// TwinCAT 3 PLC project Samples
// Title: BA2_Templates
// Company: Beckhoff Automation GmbH
// Author: Beckhoff Automation GmbH
// ProjectVersion: 2.2.0.0
// Description: Library that covers all technical building automation services in a built-in skeleton. It contains function blocks for conventional HVAC and room automation.
// ProgramVersion: 3.1.4026.20
// libraries:
//   Tc2_MDP, * (Beckhoff Automation GmbH)
//   Tc2_SerialCom, * (Beckhoff Automation GmbH)
//   Tc2_Standard, * (Beckhoff Automation GmbH)
//   Tc2_SUPS, * (Beckhoff Automation GmbH)
//   Tc2_System, * (Beckhoff Automation GmbH)
//   Tc2_Utilities, * (Beckhoff Automation GmbH)
//   Tc3_BA2, * (Beckhoff Automation GmbH)
//   Tc3_BA2_Common, * (Beckhoff Automation GmbH)
//   Tc3_BACnetRev14, * (Beckhoff Automation GmbH)
//   Tc3_DALI, * (Beckhoff Automation GmbH)
//   Tc3_Module, * (Beckhoff Automation GmbH)
//   Tc3_XBA, * (Beckhoff Automation GmbH)
// project tree:
//   / FastTask.TcTTO, PlcTask.TcTTO (not stored)
//   POUs/ DALICommunication.TcPOU, MAIN.TcPOU
//   Templates/DUTs/Enumerations/Building/ E_BA_BuildingMode.TcDUT (not stored)
//   Templates/DUTs/Enumerations/Plant/AC/ E_BA_AC_OpMod01.TcDUT (not stored), E_BA_AC_OpMod02.TcDUT, E_BA_AC_PlantStep01.TcDUT (not stored), E_BA_AC_SelSpErc.TcDUT, E_BA_AC_SeqNumber_H.TcDUT (not stored), E_BA_AC_SeqNumber_T.TcDUT (not stored)
//   Templates/DUTs/Enumerations/Process/ E_BA_Process.TcDUT (not stored)
//   Templates/DUTs/Enumerations/System/ E_BA_UPSType.TcDUT (not stored)
//   Templates/DUTs/Enumerations/Universal/ E_BA_3Point.TcDUT (not stored), E_BA_3PointA.TcDUT, E_BA_3Step.TcDUT, E_BA_3StepA.TcDUT, E_BA_Conversion_kFactor.TcDUT (not stored), E_BA_EnergyLvl.TcDUT (not stored), E_BA_EnergyLvlA.TcDUT, E_BA_EnergyLvlEx.TcDUT, E_BA_EnergyLvlExA.TcDUT, E_BA_OnOff.TcDUT, E_BA_OnOffA.TcDUT (not stored)
//   Templates/DUTs/Types/Actuator/ ST_BA_LightActuatorFeedback.TcDUT (not stored), ST_BA_SunblindActuatorFeedback.TcDUT (not stored)
//   Templates/DUTs/Types/Building/ ST_BA_BuildingAlarms.TcDUT (not stored), ST_BA_BuildingLighting.TcDUT, ST_BA_BuildingSunblind.TcDUT (not stored)
//   Templates/DUTs/Types/Facade/ ST_BA_Facade.TcDUT (not stored)
//   Templates/DUTs/Types/General/ ST_BA_GeneralSettings.TcDUT (not stored), ST_BA_GlobalAlarmsEvents.TcDUT
//   Templates/DUTs/Types/WeatherStation/ ST_BA_WeatherStation.TcDUT (not stored), ST_BA_WSC11Data.TcDUT, ST_BA_WSC11Status.TcDUT (not stored)
//   Templates/GVLs/ BA2_Param.TcGVL, LblComp.TcGVL, Priority.TcGVL (not stored), SysTime.TcGVL
//   Templates/GVLs/EventClassesID/ EC_ID.TcGVL (not stored)
//   Templates/GVLs/Language/English/ LblAggregates_EN.TcGVL, LblControl_EN.TcGVL, LblFunctions_EN.TcGVL, LblPlant_EN.TcGVL, TxtEvent_EN.TcGVL, TxtPlant_EN.TcGVL, TxtTrade_EN.TcGVL
//   Templates/GVLs/Language/German/ LblAggregates_DE.TcGVL, LblControl_DE.TcGVL, LblFunctions_DE.TcGVL, LblPlant_DE.TcGVL, TxtEvent_DE.TcGVL, TxtPlant_DE.TcGVL, TxtTrade_DE.TcGVL
//   Templates/GVLs/Site/ Site.TcGVL
//   Templates/POUs/Trade/AirConditioning/Aggregates/Cooler/Temperature/ FB_BA_AC_ColTSuACtrl.TcPOU, FB_BA_AC_ColT_02.TcPOU
//   Templates/POUs/Trade/AirConditioning/Aggregates/Damper/ FB_BA_AC_Dmp2P.TcPOU
//   Templates/POUs/Trade/AirConditioning/Aggregates/ERC/ FB_BA_AC_ErcTSuACtrl.TcPOU
//   Templates/POUs/Trade/AirConditioning/Aggregates/ERC/Plate/ FB_BA_AC_ErcPl_02.TcPOU
//   Templates/POUs/Trade/AirConditioning/Aggregates/Fan/ FB_BA_AC_FanCtl.TcPOU
//   Templates/POUs/Trade/AirConditioning/Aggregates/PreHeater/ FB_BA_AC_PreHtr.TcPOU, FB_BA_AC_PreHtrTSuACtrl.TcPOU (not stored), FB_BA_AC_TRtCtrl.TcPOU (not stored)
//   Templates/POUs/Trade/AirConditioning/ FB_BA_AirConditioning.TcPOU (not stored)
//   Templates/POUs/Trade/AirConditioning/General/ FB_BA_AC_OpMod1St.TcPOU, FB_BA_AC_PlantCmd_AHU_1st_10.TcPOU (not stored), FB_BA_AC_SeqT.TcPOU (not stored), FB_BA_AC_SumNgtCol.TcPOU (not stored)
//   Templates/POUs/Trade/AirConditioning/Plants/ FB_BA_AHU_1st_10.TcPOU (not stored)
//   Templates/POUs/Trade/AirConditioning/Setpoint/Temperature/ FB_BA_AC_TCasCtrl_01.TcPOU (not stored)
//   Templates/POUs/Trade/AutomationControl/ControlCabinet/ FB_BA_ControlCabinet.TcPOU, FB_BA_ControlCabinetBasic.TcPOU (not stored), FB_BA_ControlCabinetBasicExt.TcPOU (not stored)
//   Templates/POUs/Trade/AutomationControl/Device/BACnetSettings/ FB_BACnet_RcpList.TcPOU (not stored), FB_BA_Parameter.TcPOU (not stored)
//   Templates/POUs/Trade/AutomationControl/Device/ FB_BA_Device.TcPOU
//   Templates/POUs/Trade/AutomationControl/Device/Project/ FB_BA_ProjectEx.TcPOU
//   Templates/POUs/Trade/AutomationControl/Device/TimeSettings/ FB_BA_BACnetTime_TO_SysTime.TcPOU (not stored), FB_BA_ExternalSysTime.TcPOU
//   Templates/POUs/Trade/AutomationControl/EventClasses/ FB_BA_EvtGroups.TcPOU, FB_BA_EvtGroupsAMEV2017.TcPOU
//   Templates/POUs/Trade/AutomationControl/ FB_BA_AutomationControl.TcPOU (not stored)
//   Templates/POUs/Trade/BuildingAutomation/Communication/ FB_BA_AdsComServer_Basic.TcPOU (not stored)
//   Templates/POUs/Trade/BuildingAutomation/ FB_BA_BuildingAutomationServer.TcPOU
//   Templates/POUs/Trade/BuildingAutomation/General/ FB_BA_BuildingData.TcPOU
//   Templates/POUs/Trade/BuildingAutomation/General/Functions/ FB_BA_BuildingEnergyLevel.TcPOU, FB_BA_BuildingMode.TcPOU, FB_BA_BuildingSpRmT.TcPOU (not stored)
//   Templates/POUs/Trade/BuildingAutomation/Weather_Data/ FB_BA_WeatherData.TcPOU
//   Templates/POUs/Trade/BuildingAutomation/Weather_Data/Parameter/ FB_BA_WeatherParameter.TcPOU
//   Templates/POUs/Trade/DoorsGatesWindowsSunProtection/Communication/ FB_BA_AdsComServer_DGWS.TcPOU (not stored)
//   Templates/POUs/Trade/DoorsGatesWindowsSunProtection/ FB_BA_DGWSPServer.TcPOU (not stored)
//   Templates/POUs/Trade/HazardDetectionAlarmSystems/BurglarAlarmSystem/ FB_BA_BurglarAlarmSystem.TcPOU (not stored)
//   Templates/POUs/Trade/HazardDetectionAlarmSystems/ FB_BA_HazardDetectionAlarmSystems.TcPOU
//   Templates/POUs/Trade/HazardDetectionAlarmSystems/FireAlarmSystem/ FB_BA_FireAlarmSystem.TcPOU (not stored)
//   Templates/POUs/Trade/HeatingSystem/Distribution/HeatingCircuit/ FB_BA_H_HtgCir01.TcPOU (not stored)
//   Templates/POUs/Trade/HeatingSystem/ FB_BA_Heating.TcPOU
//   Templates/POUs/Trade/HeatingSystem/General/ FB_BA_HtgLmt.TcPOU (not stored), FB_BA_H_OpMod.TcPOU
//   Templates/POUs/Trade/HeatingSystem/Setpoint/ FB_BA_H_HtgCir_Sp.TcPOU (not stored)
//   Templates/POUs/Trade/RoomAutomation/Common/DALI FunctionBlocks/ FB_BA_BrtnsPrcDALI.TcPOU (not stored), FB_BA_LightActrDALI_Base.TcPOU, FB_BA_LightActrDALI_TC.TcPOU (not stored)
//   Templates/POUs/Trade/RoomAutomation/Common/Sensors/ FB_BA_BrightnessPresenceDALI.TcPOU
//   Templates/POUs/Trade/RoomAutomation/Communication/ FB_BA_AdsComServer_Room.TcPOU
//   Templates/POUs/Trade/RoomAutomation/ FB_BA_RoomAutomationServer.TcPOU (not stored)
//   Templates/POUs/Trade/RoomAutomation/HeatingCooling/Functions/Zone/ FB_BA_HeatCool_PID.TcPOU (not stored)
//   Templates/POUs/Trade/RoomAutomation/HeatingCooling/[Internal]/ FB_BA_Ext_HeatCoolBase.TcPOU
//   Templates/POUs/Trade/RoomAutomation/Lighting/Actuators/ FB_BA_LightAnalog.TcPOU (not stored), FB_BA_LightDALI_TC.TcPOU (not stored)
//   Templates/POUs/Trade/RoomAutomation/Lighting/Functions/Zone/ FB_BA_LightGroupConstant.TcPOU
//   Templates/POUs/Trade/RoomAutomation/Lighting/[Internal]/ FB_BA_Ext_BrightnessPresence_Base.TcPOU (not stored), FB_BA_Ext_LightBase.TcPOU (not stored), FB_BA_Ext_LightConstCtrl.TcPOU, FB_BA_Ext_LightCtrl.TcPOU (not stored)
//   Templates/POUs/Trade/RoomAutomation/RoomSamples/ FB_BA_RoomSample1.TcPOU
//   Templates/POUs/Trade/RoomAutomation/SunProtection/Actuators/ FB_BA_SunBld.TcPOU
//   Templates/POUs/Trade/RoomAutomation/SunProtection/Functions/Building/ FB_BA_BuildingSunprotection.TcPOU, FB_BA_IceProtection.TcPOU (not stored)
//   Templates/POUs/Trade/RoomAutomation/SunProtection/Functions/Facade/ FB_BA_Facade.TcPOU, FB_BA_Facade_Information.TcPOU, FB_BA_Facade_Maintenance.TcPOU, FB_BA_Facade_ParkPosition.TcPOU, FB_BA_Facade_SunProtection.TcPOU (not stored), FB_BA_Facade_ThermoAutomatic.TcPOU, FB_BA_Facade_TwilightAutomatic.TcPOU (not stored), FB_BA_Facade_WindProtection.TcPOU
//   Templates/POUs/Trade/RoomAutomation/SunProtection/Functions/Zone/ FB_BA_SunblindZone.TcPOU (not stored)
//   Templates/POUs/Trade/RoomAutomation/SunProtection/[Internal]/ FB_BA_Ext_SunblindAngle.TcPOU (not stored), FB_BA_Ext_SunblindBase.TcPOU, FB_BA_Ext_SunblindPosition.TcPOU (not stored)
//   Templates/POUs/Universal/Aggregat/Analog/ FB_BA_ActuatorAnalog.TcPOU (not stored), FB_BA_ActuatorAV.TcPOU (not stored)
//   Templates/POUs/Universal/Aggregat/Binary/ FB_BA_ActuatorCmd.TcPOU (not stored)
//   Templates/POUs/Universal/Aggregat/Modulation/ FB_BA_ActuatorMdlt.TcPOU (not stored)
//   Templates/POUs/Universal/Aggregat/Multistate/ FB_BA_ActuatorMultistate.TcPOU (not stored)
//   Templates/POUs/Universal/Control/AntiBlocking/ FB_BA_AntiBlocking.TcPOU
//   Templates/POUs/Universal/Control/EventClasses/ FB_BA_EvtCategory.TcPOU (not stored)
//   Templates/POUs/Universal/Control/Hysteresis/ FB_BA_Hys_03.TcPOU (not stored), FB_BA_Hys_21.TcPOU (not stored)
//   Templates/POUs/Universal/Control/Monitoring/ FB_BA_FdbAnalog.TcPOU (not stored), FB_BA_FdbBinary.TcPOU, FB_BA_PresenceMonitoring.TcPOU (not stored)
//   Templates/POUs/Universal/Control/Object/ FB_BA_AV_Op_SP.TcPOU, FB_BA_BV_OP_Val.TcPOU
//   Templates/POUs/Universal/Control/PID/ FB_BA_PID.TcPOU (not stored), FB_BA_PID_Sp.TcPOU (not stored)
//   Templates/POUs/Universal/Control/Ramp/ FB_BA_RampLimitIncrease.TcPOU (not stored)
//   Templates/POUs/Universal/Control/Scale/ FB_BA_Scale_02.TcPOU (not stored), FB_BA_Scale_04.TcPOU, FB_BA_Scale_04_Y2_3.TcPOU (not stored)
//   Templates/POUs/Universal/Control/TimeDelay/ FB_BA_DlyOff.TcPOU (not stored), FB_BA_DlyOn.TcPOU
//   Templates/POUs/Universal/Control/Trend/ FB_BA_TrendLogging.TcPOU
//   Templates/POUs/Universal/Motor/1st/ FB_BA_Mot1st.TcPOU (not stored)
//   Templates/POUs/Universal/Motor/Control/ FB_BA_MotCtl.TcPOU
//   Templates/POUs/Universal/Pump/1st/ FB_BA_Pu1st.TcPOU
//   Templates/POUs/Universal/Sensor/ FB_BA_CombinationBI_BV.TcPOU (not stored), FB_BA_SensorAnalog.TcPOU (not stored), FB_BA_SensorBinary.TcPOU (not stored)
//   Templates/POUs/Universal/Valve/ FB_BA_Vlv.TcPOU
//   Templates/POUs/Universal/WeatherStation/Thies/ FB_BA_ThiesData.TcPOU (not stored), FB_BA_ThiesWSC11.TcPOU (not stored), FB_BA_WeatherStation_Thies.TcPOU (not stored)
// real-time tasks:
//   TASK PlcTask: cycle T#45ms, priority 20, ADS port 350
//   TASK Device 1 (BACnet IP)_Task_58: cycle T#40ms, priority 58, ADS port 351
//   TASK Device 1 (BACnet IP)_QueueTask: cycle T#2ms, priority 8, ADS port 352
//   TASK FastTask: cycle T#5ms, priority 1, ADS port 353
// I/O:
//   DEVICE Device 1 (BACnet IP), AmsNetId 10.10.1.201.2.1
// variable links:
//   Samples/Samples Instance <-> Device 1 (BACnet IP)
//     PlcTask Inputs/BACnet_Globals.DefaultAdapter.BACnet_AmsNetId <-> Inputs/AmsNetId

CONFIGURATION Samples
    RESOURCE PLC ON TwinCAT3
        TASK FastTask(INTERVAL := T#5ms, PRIORITY := 1);
        PROGRAM DALICommunication WITH FastTask : DALICommunication;
    END_RESOURCE
END_CONFIGURATION

// ---- Templates/DUTs/Enumerations/Plant/AC/E_BA_AC_OpMod02.TcDUT
{region '#Template'}
	{attribute 'Version' := '5.0.0.0'}
	{attribute 'Tags' := '"LCID": "1031", "Text": "DUT, Enumeration, Anlage, AC, Betriebsart"'}
	{attribute 'Tags' := '"LCID": "1033", "Text": "DUT, Enumeration, Plant, AC, Operation mode"'}
	{attribute 'Description' := '"LCID": "1031", "Text": "Betriebsart Klimaanlage"'}
	{attribute 'Description' := '"LCID": "1033", "Text": "Operation mode air conditioning"'}
{endregion}

{attribute qualified_only}
TYPE E_BA_AC_OpMod02 :
(
    Invalid							:= 0,
    eOff							:= 1,	// Aus//Off
    eStep1							:= 2,	// Stufe 1						// Step 1
    eStep2							:= 3,	// Stufe 2						// Step 2
    eStep3							:= 4,	// Stufe 3						// Step 3
    eEmergency						:= 5,	// Notfall						// Emergency
    eFrost							:= 6,	// Frost						// Frost
    eSmokeExtractionProgramm		:= 7,	// Entrauchung Programm			// Smoke extraction program
    eSmokeExtractionSupplyAir		:= 8,	// Entrauchung Zuluft			// Smoke extraction supply air
    eSmokeExtractionExhaustAir		:= 9,	// Entrauchung Fortluft			// Smoke extraction exhaust air
    eFire							:= 10,	// Feuer						// Fire
    eNightCooling					:= 11,	// Nachtkühlung					// Night cooling
    eCoolDownProtection				:= 12,	// Stützbetrieb,Auskühlschutz	// Cool down protection
    eOverHeatingProtection			:= 13,	// Überhitzungsschutz			// Over heating protection
    eAlarm							:= 14,	// Störung						// Alarm
    eForcedVentilation				:= 15,	// Zwangsbelüftung				// Forced ventilation
    eCentralSwitchOff				:= 16	// Zentralabschaltung			// Central switch-off
) UDINT;
END_TYPE

// ---- Templates/DUTs/Enumerations/Plant/AC/E_BA_AC_SelSpErc.TcDUT
{region '#Template'}
	{attribute 'Version' := '5.0.0.0'}
	{attribute 'Tags' := '"LCID": "1031", "Text": "DUT, Enumeration, Anlage, AC, Sollwert"'}
	{attribute 'Tags' := '"LCID": "1033", "Text": "DUT, Enumeration, Plant, AC, Setpoint"'}
	{attribute 'Description' := '"LCID": "1031", "Text": "Auswahl Sollwert Energie Rückgewinnung"'}
	{attribute 'Description' := '"LCID": "1033", "Text": "Selection setpoint energy recovery"'}
{endregion}

{attribute 'qualified_only'}
TYPE E_BA_AC_SelSpErc :
(
	eAction				:= 1,	//	E_BA_Action.eDirect = SpCol, E_BA_Action.eReverse = SpHtg, 
	eAverageHtgCol		:= 2	
) UDINT;
END_TYPE

// ---- Templates/DUTs/Enumerations/Universal/E_BA_3PointA.TcDUT
{region '#Template'}
	{attribute 'Version' := '5.0.0.0'}
	{attribute 'Tags' := '"LCID": "1031", "Text": "DUT, Enumeration, Betriebsart, Universal, 3Point"'}
	{attribute 'Tags' := '"LCID": "1033", "Text": "DUT, Enumeration, Operation mode, Universal, 3Point"'}
	{attribute 'Description' := '"LCID": "1031", "Text": "Betriebsart 3 Punkt"'}
	{attribute 'Description' := '"LCID": "1033", "Text": "Operating mode 3 point"'}
{endregion}

{attribute 'qualified_only'}
TYPE E_BA_3PointA :
(
	eAutomatic		:= 1,
	eOff			:= 2,
	eOpen			:= 3,
	eClose			:= 4
	
) UDINT;
END_TYPE

// ---- Templates/DUTs/Enumerations/Universal/E_BA_3Step.TcDUT
{region '#Template'}
	{attribute 'Version' := '5.0.0.0'}
	{attribute 'Tags' := '"LCID": "1031", "Text": "DUT, Enumeration, Betriebsart, Universal, 3Step"'}
	{attribute 'Tags' := '"LCID": "1033", "Text": "DUT, Enumeration, Operation mode, Universal, 3Step"'}
	{attribute 'Description' := '"LCID": "1031", "Text": "Betriebsart 3 3Step"'}
	{attribute 'Description' := '"LCID": "1033", "Text": "Operating mode 3 steps"'}
{endregion}

{attribute qualified_only}
TYPE E_BA_3Step :
(
	eOff			:= 1,
	eStep1			:= 2,
	eStep2			:= 3,
	eStep3			:= 4
	
) UDINT;
END_TYPE

// ---- Templates/DUTs/Enumerations/Universal/E_BA_3StepA.TcDUT
{region '#Template'}
	{attribute 'Version' := '5.0.0.0'}
	{attribute 'Tags' := '"LCID": "1031", "Text": "DUT, Enumeration, Betriebsart, Universal, 3Step"'}
	{attribute 'Tags' := '"LCID": "1033", "Text": "DUT, Enumeration, Operation mode, Universal, 3Step"'}
	{attribute 'Description' := '"LCID": "1031", "Text": "Betriebsart 3 3Step"'}
	{attribute 'Description' := '"LCID": "1033", "Text": "Operating mode 3 steps"'}
{endregion}

{attribute qualified_only}
TYPE E_BA_3StepA :
(
	eAutomatic		:= 1,
	eOff			:= 2,
	eStep1			:= 3,
	eStep2			:= 4,
	eStep3			:= 5
	
) UDINT;
END_TYPE

// ---- Templates/DUTs/Enumerations/Universal/E_BA_EnergyLvlA.TcDUT
{region '#Template'}
	{attribute 'Version' := '5.0.0.0'}
	{attribute 'Tags' := '"LCID": "1031", "Text": "DUT, Enumeration, Room automation, Heating system"'}
	{attribute 'Tags' := '"LCID": "1033", "Text": "DUT, Enumeration, Room automation, Heating system"'}
	{attribute 'Description' := '"LCID": "1031", "Text": "Betriebsart Energieniveau"'}
	{attribute 'Description' := '"LCID": "1033", "Text": "Operating mode Energy level"'}
{endregion}

{attribute qualified_only}
TYPE E_BA_EnergyLvlA :
(
	eAutomatic		:= 1,
	eProtection		:= 2,
	eEconomy		:= 3,
	eComfort		:= 4
	
) UDINT;
END_TYPE

// ---- Templates/DUTs/Enumerations/Universal/E_BA_EnergyLvlEx.TcDUT
{region '#Template'}
	{attribute 'Version' := '5.0.0.0'}
	{attribute 'Tags' := '"LCID": "1031", "Text": "DUT, Enumeration, Room automation, Heating system"'}
	{attribute 'Tags' := '"LCID": "1033", "Text": "DUT, Enumeration, Room automation, Heating system"'}
	{attribute 'Description' := '"LCID": "1031", "Text": "Betriebsart Energieniveau"'}
	{attribute 'Description' := '"LCID": "1033", "Text": "Operating mode Energy level"'}
{endregion}

{attribute qualified_only}
TYPE E_BA_EnergyLvlEx :
(
	eProtection			:= 1,
	eEconomy			:= 2,
	ePreComfort			:= 3,
	eComfort			:= 4
	
) UDINT;
END_TYPE

// ---- Templates/DUTs/Enumerations/Universal/E_BA_EnergyLvlExA.TcDUT
{region '#Template'}
	{attribute 'Version' := '5.0.0.0'}
	{attribute 'Tags' := '"LCID": "1031", "Text": "DUT, Enumeration, Room automation, Heating system"'}
	{attribute 'Tags' := '"LCID": "1033", "Text": "DUT, Enumeration, Room automation, Heating system"'}
	{attribute 'Description' := '"LCID": "1031", "Text": "Betriebsart Energieniveau"'}
	{attribute 'Description' := '"LCID": "1033", "Text": "Operating mode Energy level"'}
{endregion}

{attribute qualified_only}
TYPE E_BA_EnergyLvlExA :
(
	eAutomatic		:= 1,
	eProtection		:= 2,
	eEconomy		:= 3,
	ePreComfort		:= 4,
	eComfort		:= 5
	
) UDINT;
END_TYPE

// ---- Templates/DUTs/Enumerations/Universal/E_BA_OnOff.TcDUT
{region '#Template'}
	{attribute 'Version' := '5.0.0.0'}
	{attribute 'Tags' := '"LCID": "1031", "Text": "DUT, Enumeration, Betriebsart, Universal, On, Off"'}
	{attribute 'Tags' := '"LCID": "1033", "Text": "DUT, Enumeration, Operation mode, Universal, On, Off"'}
	{attribute 'Description' := '"LCID": "1031", "Text": "Betriebsart Ein Aus"'}
	{attribute 'Description' := '"LCID": "1033", "Text": "Operating on off"'}
{endregion}

{attribute qualified_only}
TYPE E_BA_OnOff :
(
	eOff			:= 1,
	eOn				:= 2
	
) UDINT;
END_TYPE

// ---- Templates/DUTs/Types/Building/ST_BA_BuildingLighting.TcDUT
{region '#Template'}
	{attribute 'Version' := '5.1.0.0'}
	{attribute 'Tags' := '"LCID": "1031", "Text": "DUT, Types, Publisher, Subscriber, RA, General, Building, Lighting"'}
	{attribute 'Tags' := '"LCID": "1033", "Text": "DUT, Types, Publisher, Subscriber, RA, General, Building, Lighting"'}
	{attribute 'Description' := '"LCID": "1031", "Text": "Gebäudedaten/-status für die Raumautomation - Beleuchtung"'}
	{attribute 'Description' := '"LCID": "1033", "Text": "Building-data/-states for room-automation - Lighting"'}
{endregion}
TYPE ST_BA_BuildingLighting :
STRUCT
	stLighting 					: ST_BA_Lighting;
	bGlobalReset				: BOOL;
   {attribute 'hide'}
	aDummy						: ARRAY[1..7] OF BYTE; 		// padding bytes, in order to reach a limit corresponding to the largest data type (divisible by 8 bytes)
END_STRUCT
END_TYPE

// ---- Templates/DUTs/Types/General/ST_BA_GlobalAlarmsEvents.TcDUT
{region '#Template'}
	{attribute 'Version' := '5.0.0.0'}
	{attribute 'Tags' := '"LCID": "1031", "Text": "DUT, Types, Publisher, Subscriber, Global, General, Alarms, Events"'}
	{attribute 'Tags' := '"LCID": "1033", "Text": "DUT, Types, Publisher, Subscriber, Global, General, Alarms, Events"'}
	{attribute 'Description' := '"LCID": "1031", "Text": "Globale Alarme und Events"'}
	{attribute 'Description' := '"LCID": "1033", "Text": "Global alarms and events"'}
{endregion}
TYPE ST_BA_GlobalAlarmsEvents :
STRUCT
	bBurglary				: BOOL;
	bFireAlert				: BOOL;
	bCentralOff				: BOOL;
	bForcedVentilation		: BOOL;
	bAlarm1					: BOOL;
	bAlarm2					: BOOL;
	bAlarm3					: BOOL;
	bEvent1					: BOOL;
	bEvent2					: BOOL;
	bEvent3					: BOOL;
   {attribute 'hide'}
	aDummy					: ARRAY[1..6] OF BYTE; 		// padding bytes, in order to reach a limit corresponding to the largest data type (divisible by 8 bytes)
END_STRUCT
END_TYPE

// ---- Templates/DUTs/Types/WeatherStation/ST_BA_WSC11Data.TcDUT
{region '#Template'}
	{attribute 'Version' := '5.0.0.0'}
	{attribute 'Tags' := '"LCID": "1031", "Text": "DUT, Types, Publisher, Subscriber, Weather, Data, Thies"'}
	{attribute 'Tags' := '"LCID": "1033", "Text": "DUT, Types, Publisher, Subscriber, Weather, Data, Thies"'}
	{attribute 'Using' := '"Type": "Template", "URI": "ST_BA_WSC11Status"'}		 
	{attribute 'Description' := '"LCID": "1031", "Text": "Daten Wetterstation Thies"'}
	{attribute 'Description' := '"LCID": "1033", "Text": "Weatherstation-data Thies"'}
{endregion}
TYPE ST_BA_WSC11Data :
STRUCT
	stStatus				: ST_BA_WSC11Status;
	fCaseTemperature		: REAL;				// [°C]	 
	fLatitude				: REAL;				// [°]
	fLongitude				: REAL;				// [°]
	fSunAzimuth				: REAL;				// [°]
	fSunElevation			: REAL;				// [°]
	bRain					: BOOL;
	stDateTime				: TIMESTRUCT;
	sTimeFormat				: STRING(7);
	fOutsideTemperature		: REAL;				// [°C]
	fDewPointTemperature	: REAL;				// [°C]
	fPressureAbs			: REAL;				// [hPa]
	fPressureRel			: REAL;				// [hPa]
	fHumidityAbs			: REAL;				// [%rF]
	fHumidityRel			: REAL;				// [g/m³]
	fBrightnessNorth		: REAL;				// [kLux]
	fBrightnessEast			: REAL;				// [kLux]
	fBrightnessSouth		: REAL;				// [kLux]
	fBrightnessWest			: REAL;				// [kLux]
	fDawn					: REAL;				// [Lux] 
	fGlobalRadiation		: REAL;				// [W/m²]
	fWindDirection			: REAL;				// [°]
	fWindSpeed				: REAL;				// [m/s]
END_STRUCT
END_TYPE

// ---- Templates/GVLs/BA2_Param.TcGVL
{region '#Template'}
	{attribute 'Version' := '5.0.1.0'}
	{attribute 'Tags' := '"LCID": "1031", "Text": "GVL, Constants"'}
	{attribute 'Tags' := '"LCID": "1033", "Text": "GVL, Constants"'}
	{attribute 'Description' := '"LCID": "1031", "Text": "Globale Konstanten"'}
	{attribute 'Description' := '"LCID": "1033", "Text": "Global constants"'}
{endregion}

{attribute 'qualified_only'}
{attribute 'strict'}
VAR_GLOBAL CONSTANT 
	fAP                					: REAL 						:= 1013.25;	// Hydrostatischer Luftdruck	//	atmospheric pressure

	nDefTimeDelay_ToAbnormal			: UDINT						:= 1;
	nDefTimeDelay_ToNormal				: UDINT						:= 1;

	fDefCOVIncrement					: REAL						:= 0.1;	

	fDefLimitDeadband					: REAL						:= 0.0;

	nLoop_DefOpMode						: E_BA_PIDMode				:= E_BA_PIDMode.eP1ID;	
	
	stTrend_DefStartTime				: ST_BA_DateTime			:= ();
	stTrend_DefStopTime					: ST_BA_DateTime			:= ();
	
	nTrend_BufferSize					: UDINT						:= 500;	// Count of entries in a Trend-Buffer	
	bTrend_DefLogEnable					: BOOL						:= FALSE;
	bTrend_DefStopOnFull				: BOOL						:= FALSE;
	nTrend_DefLogInterval				: UDINT						:= 90;	// (in [s])
	nTrend_DefNotificationThreshold		: UDINT						:= 50;
	eTrend_DefLoggingType				: E_BA_LoggingType			:= E_BA_LoggingType.ePolled;			
	
	nMaxNumberOfFacades					: USINT:=4;
	nMaxNumberOfAreas					: USINT:=4;
END_VAR
VAR_GLOBAL
	bBlink								: BOOL;
	bDlyStartPLC						: BOOL 						:= TRUE;	
END_VAR

// ---- Templates/GVLs/Language/English/LblAggregates_EN.TcGVL
{region '#Template'}
	{attribute 'Version' := '5.2.0.0'}
	{attribute 'Tags' := '"LCID": "1031", "Text": "GVL, AKS, Labels, ObjectName, Description"'}
	{attribute 'Tags' := '"LCID": "1033", "Text": "GVL, DPAD, Labels, ObjectName, Description"'}
	{attribute 'Description' := '"LCID": "1031", "Text": "Anlagenkennzeichnungssystem, Labels Aggregate"'}
	{attribute 'Description' := '"LCID": "1033", "Text": "Data Point Addressing Description, Labels aggregate"'}
{endregion}
	 
{attribute 'global_init_slot' := '40510'}
VAR_GLOBAL
  LblAgg_FunctionallyIndependentEequipment                 :FB_BA_Label:=( sObjName:='FIE',sDescr:='Functionally independent equipment');
  LblAgg_SelfContainedControlUnit                          :FB_BA_Label:=( sObjName:='SCR',sDescr:='Self-contained control or regulation unit');
  LblAgg_ControlCabinet                                    :FB_BA_Label:=( sObjName:='CCB',sDescr:='Control cabinet (trade-specific)');
//     330 Doors, gates, windows, sun protection
  LblAgg_WindowDrive                                       :FB_BA_Label:=( sObjName:='WIN',sDescr:='Window (drive)');
  LblAgg_WindowContact                                     :FB_BA_Label:=( sObjName:='WIC',sDescr:='Window contact');
  LblAgg_Blind                                             :FB_BA_Label:=( sObjName:='BLD',sDescr:='Blind');
  LblAgg_Awning                                            :FB_BA_Label:=( sObjName:='AWN',sDescr:='Awning');
  LblAgg_RollerShutters                                    :FB_BA_Label:=( sObjName:='ROS',sDescr:='Roller shutters');
  LblAgg_Gate                                              :FB_BA_Label:=( sObjName:='GAT',sDescr:='Gate');
  LblAgg_Door                                              :FB_BA_Label:=( sObjName:='DOR',sDescr:='Door');
  LblAgg_DoorContact                                       :FB_BA_Label:=( sObjName:='DOC',sDescr:='Door contact');
  LblAgg_Blackout                                          :FB_BA_Label:=( sObjName:='BLA',sDescr:='Blackout');
//     412 Water plants
  LblAgg_TraceHeating                                      :FB_BA_Label:=( sObjName:='THT',sDescr:='Trace heating');
  LblAgg_ElectricHeating                                   :FB_BA_Label:=( sObjName:='EHT',sDescr:='Electric heating (warm water temperature preparation)');
  LblAgg_WaterFilter                                       :FB_BA_Label:=( sObjName:='WFL',sDescr:='Water filter');
//     421 Heat generation plants
  LblAgg_Furnace                                           :FB_BA_Label:=( sObjName:='FUR',sDescr:='Furnace');
  LblAgg_HeatExchanger                                     :FB_BA_Label:=( sObjName:='HEX',sDescr:='Heat exchanger');
//     430 Ventilation and refrigeration systems
  LblAgg_FanExhaustAir                                     :FB_BA_Label:=( sObjName:='EHF',sDescr:='Exhaust air fan');
  LblAgg_Airwasher                                         :FB_BA_Label:=( sObjName:='AWA',sDescr:='Airwasher');
  LblAgg_Humidifier                                        :FB_BA_Label:=( sObjName:='HUF',sDescr:='Humidifier');
  LblAgg_HumidifierPump                                    :FB_BA_Label:=( sObjName:='HUP',sDescr:='Humidifier pump');
  LblAgg_FireDamper                                        :FB_BA_Label:=( sObjName:='FID',sDescr:='Fire damper, fire protection valve');
  LblAgg_SmokeProtectionDamper                             :FB_BA_Label:=( sObjName:='SPD',sDescr:='Smoke protection damper');
  LblAgg_SmokeExtractorDamper                              :FB_BA_Label:=( sObjName:='SEP',sDescr:='Smoke extractor damper');
  LblAgg_CeilingSwirlDiffuser                              :FB_BA_Label:=( sObjName:='CSD',sDescr:='Ceiling swirl diffuser');
  LblAgg_RoofAirHeater                                     :FB_BA_Label:=( sObjName:='RAH',sDescr:='Roof air heater');
  LblAgg_DirectEvaporator                                  :FB_BA_Label:=( sObjName:='DEA',sDescr:='Direct evaporator');
  LblAgg_ElectricalAirHeater                               :FB_BA_Label:=( sObjName:='EAH',sDescr:='Electrical air heater');
  LblAgg_ElectricReHeater                                  :FB_BA_Label:=( sObjName:='ERH',sDescr:='Electric re-heater');
  LblAgg_ElectricaPreHeater                                :FB_BA_Label:=( sObjName:='EPH',sDescr:='Electrical pre-heater');
  LblAgg_HeaterGeneral                                     :FB_BA_Label:=( sObjName:='HTR',sDescr:='Heater ');
  LblAgg_FanExtractAir                                     :FB_BA_Label:=( sObjName:='EXF',sDescr:='Extract air fan ');
  LblAgg_InductionDevice                                   :FB_BA_Label:=( sObjName:='IND',sDescr:='Induction device');
  LblAgg_RefrigerantDryer                                  :FB_BA_Label:=( sObjName:='RFD',sDescr:='Refrigerant dryer');
  LblAgg_CirculatorySystem                                 :FB_BA_Label:=( sObjName:='CCS',sDescr:='Circulatory system ');
  LblAgg_AirFilterOutsideAir                               :FB_BA_Label:=( sObjName:='AFI',sDescr:='Outside air filter');
  LblAgg_AirFilterSupplyAir                                :FB_BA_Label:=( sObjName:='AFI',sDescr:='Supply air filter');
  LblAgg_AirFilterExhaustAir                               :FB_BA_Label:=( sObjName:='AFI',sDescr:='Exhaus air filter');
  LblAgg_AirFilterExtractAir                               :FB_BA_Label:=( sObjName:='AFI',sDescr:='Extract air filter');
  LblAgg_AirFilter                                         :FB_BA_Label:=( sObjName:='AFI',sDescr:='Air filter');
  LblAgg_VentilationDamper                                 :FB_BA_Label:=( sObjName:='VFL',sDescr:='Ventilation flap');
  LblAgg_VentilationDamperOutsideAir                       :FB_BA_Label:=( sObjName:='VFL',sDescr:='Ventilation flap outside air');
  LblAgg_VentilationDamperExhaustAir                       :FB_BA_Label:=( sObjName:='VFL',sDescr:='Ventilation flap exhaust air');
  LblAgg_VentilationDamperMixAir                           :FB_BA_Label:=( sObjName:='VFL',sDescr:='Ventilation flap mix air');
  LblAgg_VentilationDamperSupplyAir                        :FB_BA_Label:=( sObjName:='VFL',sDescr:='Ventilation flap supply air');
  LblAgg_VentilationDamperBypassAir                        :FB_BA_Label:=( sObjName:='VFL',sDescr:='Ventilation flap bypass');
  LblAgg_Pump                                              :FB_BA_Label:=( sObjName:='PUM',sDescr:='Pump');
  LblAgg_RecirculatingAirCoolingDevice                     :FB_BA_Label:=( sObjName:='RAC',sDescr:='Recirculating air cooling device');
  LblAgg_FanRecirculatingAir                               :FB_BA_Label:=( sObjName:='RAF',sDescr:='Recirculating air fan');
  LblAgg_UvFilter                                          :FB_BA_Label:=( sObjName:='UVF',sDescr:='UV filter');
  LblAgg_VariableFlowRateController                        :FB_BA_Label:=( sObjName:='VFC',sDescr:='Variable flow rate controller');
  LblAgg_WaterAirHeater                                    :FB_BA_Label:=( sObjName:='WAH',sDescr:='Water air heater');
  LblAgg_WaterReHeater                                     :FB_BA_Label:=( sObjName:='WRH',sDescr:='Water re-heater');
  LblAgg_WaterPreHeater                                    :FB_BA_Label:=( sObjName:='WPH',sDescr:='Water pre-heater');
  LblAgg_HeatRecovery                                      :FB_BA_Label:=( sObjName:='HRC',sDescr:='Heat recovery');
  LblAgg_FanSupplyAir                                      :FB_BA_Label:=( sObjName:='SUF',sDescr:='Supply air fan');
  LblAgg_SmokeExtractionSystems                            :FB_BA_Label:=( sObjName:='SES',sDescr:='Smoke extraction systems');
  LblAgg_SmokeExtractionVentilator                         :FB_BA_Label:=( sObjName:='SEF',sDescr:='Smoke extraction fan');
  LblAgg_VentWindow                                        :FB_BA_Label:=( sObjName:='VWI',sDescr:='Vent window');
  LblAgg_VentFlap                                          :FB_BA_Label:=( sObjName:='VFL',sDescr:='Vent flap');
  LblAgg_VentDoor                                          :FB_BA_Label:=( sObjName:='VDO',sDescr:='Vent door');
  LblAgg_WakeFan                                           :FB_BA_Label:=( sObjName:='WAF',sDescr:='Wake fan');
//     434 Refrigeration systems
  LblAgg_GlycoOilProtector                                 :FB_BA_Label:=( sObjName:='GLP',sDescr:='Glycol/oil protector');
  LblAgg_Chiller                                           :FB_BA_Label:=( sObjName:='CHI',sDescr:='Chiller');
  LblAgg_ReCoolingPlant                                    :FB_BA_Label:=( sObjName:='RCP',sDescr:='Re-cooling plant');
//     440 High-voltage systems
  LblAgg_GeneralPowerSupply                                :FB_BA_Label:=( sObjName:='GPS',sDescr:='General power supply');
  LblAgg_CombindeHeatPowerStation                          :FB_BA_Label:=( sObjName:='CGU',sDescr:='Co-generation unit');
  LblAgg_CompensationSystem                                :FB_BA_Label:=( sObjName:='CPS',sDescr:='Compensation system');
  LblAgg_CouplingSwitch                                    :FB_BA_Label:=( sObjName:='COS',sDescr:='Coupling switch');
  LblAgg_LoadBreakSwitch                                   :FB_BA_Label:=( sObjName:='LBS',sDescr:='Load-break switch');
  LblAgg_CircuitBreaker                                    :FB_BA_Label:=( sObjName:='CCB',sDescr:='Circuit breaker');
  LblAgg_NetworkAnalyser                                   :FB_BA_Label:=( sObjName:='NWA',sDescr:='Network analyser');
  LblAgg_EmergencyPoweGeneratorUnit                        :FB_BA_Label:=( sObjName:='EPG',sDescr:='Emergency power generator unit');
  LblAgg_EmergencyLighting                                 :FB_BA_Label:=( sObjName:='EML',sDescr:='Emergency lighting');
  LblAgg_SafetyPowerSupply                                 :FB_BA_Label:=( sObjName:='SPS',sDescr:='Safety power supply');
  LblAgg_Transformer                                       :FB_BA_Label:=( sObjName:='TRF',sDescr:='Transformer');
  LblAgg_UninterruptiblePowerSupply                        :FB_BA_Label:=( sObjName:='UPS',sDescr:='Uninterruptible power supply');
//     450 Telecommunications and information technology equipment
  LblAgg_CentralFireAlarmSystem                            :FB_BA_Label:=( sObjName:='CFA',sDescr:='Central fire alarm system');
  LblAgg_FireControlPanel                                  :FB_BA_Label:=( sObjName:='FCP',sDescr:='Fire control panel');
  LblAgg_KitchenTableau                                    :FB_BA_Label:=( sObjName:='KIT',sDescr:='Kitchen tableau');
  LblAgg_SmokeDetector                                     :FB_BA_Label:=( sObjName:='SDE',sDescr:='Smoke detector');
  LblAgg_SmokeProtectionScreen                             :FB_BA_Label:=( sObjName:='SPS',sDescr:='Smoke protection screen');
  LblAgg_VoiceAlarmCentre                                  :FB_BA_Label:=( sObjName:='VAC',sDescr:='Voice alarm centre');
  LblAgg_Tableau                                           :FB_BA_Label:=( sObjName:='TAB',sDescr:='Tableau (general)');
//     460 Conveyors
  LblAgg_LiftGeneral                                       :FB_BA_Label:=( sObjName:='LIG',sDescr:='Lift general');
  LblAgg_GoodsLift                                         :FB_BA_Label:=( sObjName:='GLI',sDescr:='Goods lift');
  LblAgg_PassengerLift                                     :FB_BA_Label:=( sObjName:='PLI',sDescr:='Passenger lift');
//     470 User-specific systems
  LblAgg_FumeCupboard                                      :FB_BA_Label:=( sObjName:='FCB',sDescr:='Fume cupboard');
  LblAgg_Compressor                                        :FB_BA_Label:=( sObjName:='COM',sDescr:='Compressor');
  LblAgg_ProgrammableLogicControllers                      :FB_BA_Label:=( sObjName:='PLC',sDescr:='Programmable logic controllers');
//     479 User-specific system, weather station
  LblAgg_RainSensor                                        :FB_BA_Label:=( sObjName:='RAS',sDescr:='Rain sensor');
  LblAgg_SolarRadiation                                    :FB_BA_Label:=( sObjName:='SOR',sDescr:='Solar radiation');
  LblAgg_WeatherStation                                    :FB_BA_Label:=( sObjName:='WST',sDescr:='Weather station');
  LblAgg_WindSpeed                                         :FB_BA_Label:=( sObjName:='WIS',sDescr:='Wind speed');
  LblAgg_WindDirection                                     :FB_BA_Label:=( sObjName:='WID',sDescr:='Wind direction');
  LblAgg_WindForce                                         :FB_BA_Label:=( sObjName:='WDF',sDescr:='Wind force');
  LblAgg_Brightness                                        :FB_BA_Label:=( sObjName:='BIN',sDescr:='Brightness');
  LblAgg_Dawn                                              :FB_BA_Label:=( sObjName:='BID',sDescr:='Brightness dawn');
  LblAgg_PressureAbsolute                                  :FB_BA_Label:=( sObjName:='PAB',sDescr:='Pressure absolute');
  LblAgg_PressureRelative                                  :FB_BA_Label:=( sObjName:='PRE',sDescr:='Pressure relative');
  LblAgg_GeoLatitude                                       :FB_BA_Label:=( sObjName:='LAT',sDescr:='Latitude');
  LblAgg_GeoLongitude                                      :FB_BA_Label:=( sObjName:='LOT',sDescr:='Longitude');
  LblAgg_SunAzimuth                                        :FB_BA_Label:=( sObjName:='AZI',sDescr:='Azimuth');
  LblAgg_SunElevation                                      :FB_BA_Label:=( sObjName:='ELE',sDescr:='Elevation');
  LblAgg_WeatherStationReset                               :FB_BA_Label:=( sObjName:='PLS',sDescr:='Weather station reset');
  LblAgg_WeatherStationCommReset                           :FB_BA_Label:=( sObjName:='PLS',sDescr:='Weather station reset serial communication');
  LblAgg_WeatherStationComm                                :FB_BA_Label:=( sObjName:='WST',sDescr:='Weather station communication');
//     480 Building automation and control systems
  LblAgg_SystemSwitch                                      :FB_BA_Label:=( sObjName:='SYS',sDescr:='System switch');
  LblAgg_AutomationStationEquipment                        :FB_BA_Label:=( sObjName:='ASE',sDescr:='Automation station equipment');
  LblAgg_BusLineCoupler                                    :FB_BA_Label:=( sObjName:='BUS',sDescr:='Bus line coupler');
  LblAgg_DataInterfaceUnit                                 :FB_BA_Label:=( sObjName:='DIU',sDescr:='Data interface unit');
  LblAgg_FieldbusModule                                    :FB_BA_Label:=( sObjName:='FBM',sDescr:='Fieldbus module');
  LblAgg_InformationFocalPoint                             :FB_BA_Label:=( sObjName:='IFP',sDescr:='Information focal point');
  LblAgg_ManagementAndControlEquipment                     :FB_BA_Label:=( sObjName:='MCE',sDescr:='Management and control equipment');
//     481 BACS sensors – temperature
  LblAgg_TemperatureGasEmission                            :FB_BA_Label:=( sObjName:='TEG',sDescr:='Emissions gas temperature');
  LblAgg_TemperatureExtractAir                             :FB_BA_Label:=( sObjName:='TEX',sDescr:='Extract air temperature');
  LblAgg_TemperatureOutside                                :FB_BA_Label:=( sObjName:='TOU',sDescr:='Outside temperature');
  LblAgg_TemperatureExhaustAir                             :FB_BA_Label:=( sObjName:='TEH',sDescr:='Exhaust air temperature');
  LblAgg_FrostProtectionMonitor                            :FB_BA_Label:=( sObjName:='FPM',sDescr:='Frost protection monitor');
  LblAgg_TemperatureMixedAir                               :FB_BA_Label:=( sObjName:='TMI',sDescr:='Mixed air temperature');
  LblAgg_TemperatureRoomAir                                :FB_BA_Label:=( sObjName:='TRO',sDescr:='Room temperature');
  LblAgg_TemperatureReturnFlow                             :FB_BA_Label:=( sObjName:='TRT',sDescr:='Return flow temperature');
  LblAgg_LimiterSafetyTemperature                          :FB_BA_Label:=( sObjName:='STL',sDescr:='Safety temperature limiter');
  LblAgg_MonitorSafetyTemperature                          :FB_BA_Label:=( sObjName:='STM',sDescr:='Safety temperature monitor');
  LblAgg_TemperatureStorage                                :FB_BA_Label:=( sObjName:='TST',sDescr:='Storage temperature');
  LblAgg_TemperatureDewPoint                               :FB_BA_Label:=( sObjName:='TDP',sDescr:='Dew point temperature');
  LblAgg_MonitorDewPoint                                   :FB_BA_Label:=( sObjName:='DPM',sDescr:='Dew point monitor');
  LblAgg_TemperatureAfterCooler                            :FB_BA_Label:=( sObjName:='TAC',sDescr:='Temperature after cooler');
  LblAgg_TemperatureAfterPreHeater                         :FB_BA_Label:=( sObjName:='TAP',sDescr:='Temperature after pre-heater');
  LblAgg_TemperatureAfterHeatRecovery                      :FB_BA_Label:=( sObjName:='TAR',sDescr:='Temperature after heat recovery');
  LblAgg_Thermostat                                        :FB_BA_Label:=( sObjName:='THM',sDescr:='Thermostat');
  LblAgg_TemperatureHotWater                               :FB_BA_Label:=( sObjName:='THW',sDescr:='Hot water temperature');
  LblAgg_TemperatureCirculation                            :FB_BA_Label:=( sObjName:='TCI',sDescr:='Circulation temperature');
  LblAgg_TemperatureRecirculatingAir                       :FB_BA_Label:=( sObjName:='TRE',sDescr:='Recirculating air temperature');
  LblAgg_TemperatureFlow                                   :FB_BA_Label:=( sObjName:='TFL',sDescr:='Flow temperature');
  LblAgg_TemperatureSupplyAir                              :FB_BA_Label:=( sObjName:='TSU',sDescr:='Supply air temperature');
  LblAgg_TemperatureWetBulp                                :FB_BA_Label:=( sObjName:='TWB',sDescr:='Wet bulp temperature');
  LblAgg_TemperatureWetBulpExtractAir                      :FB_BA_Label:=( sObjName:='WEX',sDescr:='Wet bulp temperature extract air');
  LblAgg_TemperatureWetBulpExhaustAir                      :FB_BA_Label:=( sObjName:='WEH',sDescr:='Wet bulp temperature exhaust air');
  LblAgg_TemperatureWetBulpOutsideAir                      :FB_BA_Label:=( sObjName:='WOU',sDescr:='Wet bulp temperature outside air');
  LblAgg_TemperatureWetBulpRoomAir                         :FB_BA_Label:=( sObjName:='WRO',sDescr:='Wet bulp temperature room air');
  LblAgg_TemperatureWetBulpSupplyAir                       :FB_BA_Label:=( sObjName:='WSU',sDescr:='Wet bulp temperature supply air');
  LblAgg_TemperatureDewPointExtractAir                     :FB_BA_Label:=( sObjName:='DEX',sDescr:='Dew point temperature extract air');
  LblAgg_TemperatureDewPointExhaustAir                     :FB_BA_Label:=( sObjName:='DEH',sDescr:='Dew point temperature exhaust air');
  LblAgg_TemperatureDewPointOutsideAir                     :FB_BA_Label:=( sObjName:='DOU',sDescr:='Dew point temperature outside air');
  LblAgg_TemperatureDewPointRoomAir                        :FB_BA_Label:=( sObjName:='DRO',sDescr:='Dew point temperature room air');
  LblAgg_TemperatureDewPointSupplyAir                      :FB_BA_Label:=( sObjName:='DSU',sDescr:='Dew point temperature supply air');
//     481 BACS sensors – pressure
  LblAgg_PressureExtractAir                                :FB_BA_Label:=( sObjName:='PEX',sDescr:='Extract air pressure');
  LblAgg_PressureOutsideAir                                :FB_BA_Label:=( sObjName:='POU',sDescr:='Outside air pressure');
  LblAgg_PressureDifferential                              :FB_BA_Label:=( sObjName:='PDI',sDescr:='Differential pressure');
  LblAgg_PressureDifferentialOutsideAirFilter              :FB_BA_Label:=( sObjName:='PDI',sDescr:='Differential pressure outside air filter');
  LblAgg_PressureDifferentialExtractAirFilter              :FB_BA_Label:=( sObjName:='PDI',sDescr:='Differential pressure extract air filter');
  LblAgg_PressureDifferentialExhaustAirFilter              :FB_BA_Label:=( sObjName:='PDI',sDescr:='Differential pressure exhaust air filter');
  LblAgg_PressureDifferentialSupplyAirFan                  :FB_BA_Label:=( sObjName:='PDI',sDescr:='Differential pressure supply air fan');
  LblAgg_PressureDifferentialExtractAirFan                 :FB_BA_Label:=( sObjName:='PDI',sDescr:='Differential pressure ectract air fan');
  LblAgg_PressureDifferentialExhaustAirFan                 :FB_BA_Label:=( sObjName:='PDI',sDescr:='Differential pressure exhaust air fan');
  LblAgg_PressureSensorFlow                                :FB_BA_Label:=( sObjName:='PFL',sDescr:='Pressure sensor (water) flow');
  LblAgg_MonitorPressure                                   :FB_BA_Label:=( sObjName:='PCO',sDescr:='Pressure controller');
  LblAgg_PressureExhaustAir                                :FB_BA_Label:=( sObjName:='PEH',sDescr:='Exhaust air pressure');
  LblAgg_PressureRoomAir                                   :FB_BA_Label:=( sObjName:='PRO',sDescr:='Room pressure');
  LblAgg_PressureIndexCircuitSensorDifferential            :FB_BA_Label:=( sObjName:='PSI',sDescr:='Index circuit sensor differential pressure');
  LblAgg_LimiterSafetyPressure                             :FB_BA_Label:=( sObjName:='SPL',sDescr:='Safety pressure limiter');
  LblAgg_PressureSupplyAir                                 :FB_BA_Label:=( sObjName:='PSU',sDescr:='Supply air pressure');
//     481 BACS sensors – air quality
  LblAgg_CO2Sensor                                         :FB_BA_Label:=( sObjName:='COM',sDescr:='CO2 sensor');
  LblAgg_CO2ExtractAir                                     :FB_BA_Label:=( sObjName:='CEX',sDescr:='Extract air CO2');
  LblAgg_CO2ExhaustAir                                     :FB_BA_Label:=( sObjName:='CEH',sDescr:='Exhaust air CO2');
  LblAgg_CO2OutsideAir                                     :FB_BA_Label:=( sObjName:='COU',sDescr:='Outside air CO2');
  LblAgg_CO2RoomAir                                        :FB_BA_Label:=( sObjName:='CRO',sDescr:='Room air CO2');
  LblAgg_CO2SupplyAir                                      :FB_BA_Label:=( sObjName:='CSU',sDescr:='Supply air CO2');
  LblAgg_QualityExtractAir                                 :FB_BA_Label:=( sObjName:='QEX',sDescr:='Extract air quality');
  LblAgg_QualityExhaustAir                                 :FB_BA_Label:=( sObjName:='QEH',sDescr:='Exhaust air quality');
  LblAgg_QualityOutsideAir                                 :FB_BA_Label:=( sObjName:='QOU',sDescr:='Outside air quality');
  LblAgg_OualityRoomAir                                    :FB_BA_Label:=( sObjName:='QRO',sDescr:='Room air quality');
  LblAgg_QualitiySupplyAir                                 :FB_BA_Label:=( sObjName:='QSU',sDescr:='Supply air quality');
  LblAgg_QualityAirSensor                                  :FB_BA_Label:=( sObjName:='AQS',sDescr:='Air quality sensor');
//     481 BACS sensors – humidity
  LblAgg_Hygrostat                                         :FB_BA_Label:=( sObjName:='HYG',sDescr:='Hygrostat');
  LblAgg_RelativeHumidityExtractAir                        :FB_BA_Label:=( sObjName:='HEX',sDescr:='Relative extract air humidity');
  LblAgg_RelativeHumidityOutsideAir                        :FB_BA_Label:=( sObjName:='HOU',sDescr:='Relative outside air humidity');
  LblAgg_RelativeHumidityExhaustAir                        :FB_BA_Label:=( sObjName:='HEH',sDescr:='Relative exhaust air humidity');
  LblAgg_MonitorCondensation                               :FB_BA_Label:=( sObjName:='HCM',sDescr:='Condensation monitor');
  LblAgg_RelativeHumidityMixedAir                          :FB_BA_Label:=( sObjName:='HMI',sDescr:='Relative mixed air humidity');
  LblAgg_RelativeHumidityRoomHumidity                      :FB_BA_Label:=( sObjName:='HRO',sDescr:='Relative room humidity');
  LblAgg_RelativeHumidityRecirculatedAir                   :FB_BA_Label:=( sObjName:='HRE',sDescr:='Relative recirculated air humidity');
  LblAgg_RelativeHumiditySupplyAir                         :FB_BA_Label:=( sObjName:='HSU',sDescr:='Relative supply air humidity');
  LblAgg_AbsoluteHumidityExtractAir                        :FB_BA_Label:=( sObjName:='XEX',sDescr:='Absolute extract air humidity');
  LblAgg_AbsoluteHumidityOutsideAir                        :FB_BA_Label:=( sObjName:='XOU',sDescr:='Absolute outsie air humidity');
  LblAgg_AbsoluteHumidityExhaustAir                        :FB_BA_Label:=( sObjName:='XEH',sDescr:='Absolute exhaust air humidity');
  LblAgg_AbsoluteHumidityMixedAir                          :FB_BA_Label:=( sObjName:='XMI',sDescr:='Absolute mixed air humidity');
  LblAgg_AbsoluteHumidityRoomAir                           :FB_BA_Label:=( sObjName:='XRO',sDescr:='Absolute room humidity');
  LblAgg_AbsoluteHumidityRecirculatingAir                  :FB_BA_Label:=( sObjName:='XRE',sDescr:='Absolute recirculating air humidity');
  LblAgg_AbsoluteHumiditySupplyAir                         :FB_BA_Label:=( sObjName:='XSU',sDescr:='Absolute supply air humidity');
//     481 BACS sensors – consumption recording
  LblAgg_MeterElectric                                     :FB_BA_Label:=( sObjName:='ELM',sDescr:='Electric meter');
  LblAgg_MeterGasNaturalGas                                :FB_BA_Label:=( sObjName:='GAM',sDescr:='Gas meter natural gas');
  LblAgg_MeterCoolingEnergy                                :FB_BA_Label:=( sObjName:='CEM',sDescr:='Cooling energy meter');
  LblAgg_MeterHeat                                         :FB_BA_Label:=( sObjName:='HEM',sDescr:='Heat meter');
  LblAgg_MetferWater                                       :FB_BA_Label:=( sObjName:='WAM',sDescr:='Water meter');
  LblAgg_MeterFuel                                         :FB_BA_Label:=( sObjName:='FUM',sDescr:='Fuel meter (oil)');
  LblAgg_MeterSteam                                        :FB_BA_Label:=( sObjName:='STM',sDescr:='Steam meter');
  LblAgg_DegreeDayNumber                                   :FB_BA_Label:=( sObjName:='DDN',sDescr:='Degree day number');
//     481 BACS sensors – condition recording and other
  LblAgg_LeakageMonitoring                                 :FB_BA_Label:=( sObjName:='LKM',sDescr:='Leakage monitoring');
  LblAgg_EmergencyStop                                     :FB_BA_Label:=( sObjName:='EMG',sDescr:='Emergency stop unit/button');
  LblAgg_StockLevel                                        :FB_BA_Label:=( sObjName:='SLV',sDescr:='Stock level');
  LblAgg_FlowMonitor                                       :FB_BA_Label:=( sObjName:='FLM',sDescr:='Flow monitor');
  LblAgg_OverflowMonitoring                                :FB_BA_Label:=( sObjName:='OVM',sDescr:='Overflow monitoring');
  LblAgg_LowWaterCutOff                                    :FB_BA_Label:=( sObjName:='WCO',sDescr:='Low-water cut-off');
  LblAgg_WaterFlowMonitor                                  :FB_BA_Label:=( sObjName:='WFM',sDescr:='Water flow monitor');
//     481 BACS sensors – speed
  LblAgg_PumpSpeed                                         :FB_BA_Label:=( sObjName:='SPU',sDescr:='Pump speed');
  LblAgg_FanSpeedExtractAir                                :FB_BA_Label:=( sObjName:='SEX',sDescr:='Fan speed (extract air)');
  LblAgg_FanSpeedExhaustAir                                :FB_BA_Label:=( sObjName:='SEH',sDescr:='Fan speed (exhaust air)');
  LblAgg_FanSpeedSupplyAir                                 :FB_BA_Label:=( sObjName:='SSU',sDescr:='Fan speed (supply air)');
//     481 BACS sensors – volume flow
  LblAgg_VolumeFlowRateExtractAir                          :FB_BA_Label:=( sObjName:='VEX',sDescr:='Extract air volume flow rate');
  LblAgg_VolumeFlowRateOutsideAir                          :FB_BA_Label:=( sObjName:='VOU',sDescr:='Outside air volume flow rate');
  LblAgg_VolumeFlowRateExhaustAir                          :FB_BA_Label:=( sObjName:='VEH',sDescr:='Exhaust air volume flow rate');
  LblAgg_VolumeFlowRateBrineCirculatorySystem              :FB_BA_Label:=( sObjName:='VBR',sDescr:='Volume flow brine (circulatory system)');
  LblAgg_VolumeFlowRateColdDrinkingWater                   :FB_BA_Label:=( sObjName:='VCW',sDescr:='Volume flow cold drinking water');
  LblAgg_VolumeFlowRateHotDrinkingWater                    :FB_BA_Label:=( sObjName:='VHW',sDescr:='Volume flow hot drinking water');
  LblAgg_VolumeFlowRateWaterPurification                   :FB_BA_Label:=( sObjName:='VWP',sDescr:='Volume flow water purification');
  LblAgg_VolumeFlowRateSupplyAir                           :FB_BA_Label:=( sObjName:='VSU',sDescr:='Supply air volume flow');
//     481 BACS senors – enthalpy
  LblAgg_Enthalpy                                          :FB_BA_Label:=( sObjName:='ETH',sDescr:='Enthalpy');
  LblAgg_EnthalpyExtractAir                                :FB_BA_Label:=( sObjName:='EEX',sDescr:='Enthalpy extract air');
  LblAgg_EnthalpyExhaustAir                                :FB_BA_Label:=( sObjName:='EEH',sDescr:='Enthalpy exhaust air');
  LblAgg_EnthalpyOutsideAir                                :FB_BA_Label:=( sObjName:='EOU',sDescr:='Enthalpy outside air');
  LblAgg_EnthalpyRoomAir                                   :FB_BA_Label:=( sObjName:='ERO',sDescr:='Enthalpy room air');
  LblAgg_EnthalpySupplyAir                                 :FB_BA_Label:=( sObjName:='ESU',sDescr:='Enthalpy supply air');
//     481 BACS senors – multifunctional sensor
  LblAgg_MultiSensorExtractAir                             :FB_BA_Label:=( sObjName:='MEX',sDescr:='Multifunctional sensor extract air');
  LblAgg_MultiSensorExhaustAir                             :FB_BA_Label:=( sObjName:='MEH',sDescr:='Multifunctional sensor exhaust air');
  LblAgg_MultiSensorOutsideAir                             :FB_BA_Label:=( sObjName:='MOU',sDescr:='Multifunctional sensor outside air');
  LblAgg_MultiSensorRoomAir                                :FB_BA_Label:=( sObjName:='MRO',sDescr:='Multifunctional sensor room air');
  LblAgg_MultiSensorSupplyAir                              :FB_BA_Label:=( sObjName:='MSU',sDescr:='Multifunctional sensor supply air');
//     481 BACS actuators – actuating drives
  LblAgg_ValveRadiator                                     :FB_BA_Label:=( sObjName:='RDV',sDescr:='Radiator valve drive');
  LblAgg_ValveCoolingCeiling                               :FB_BA_Label:=( sObjName:='CCV',sDescr:='Cooling ceiling valve drive');
  LblAgg_MotorisedFlap                                     :FB_BA_Label:=( sObjName:='FLA',sDescr:='Motorised flap');
  LblAgg_Valve                                             :FB_BA_Label:=( sObjName:='VLV',sDescr:='Motor valve');
  LblAgg_HumidifierValve                                   :FB_BA_Label:=( sObjName:='VLV',sDescr:='Humidifier valve');
//     481 BACS lighting
  LblAgg_IlluminationExternal                              :FB_BA_Label:=( sObjName:='EOU',sDescr:='Illumination outside');
  LblAgg_IlluminationRoom                                  :FB_BA_Label:=( sObjName:='ERO',sDescr:='Illumination room');
  LblAgg_LightColourRoom                                   :FB_BA_Label:=( sObjName:='CRO',sDescr:='Light colour room');
  LblAgg_RedLightIntensity                                 :FB_BA_Label:=( sObjName:='LRD',sDescr:='Red light intensity');
  LblAgg_GreenLightIntensity                               :FB_BA_Label:=( sObjName:='LGN',sDescr:='Green light intensity');
  LblAgg_BlueLightIntensity                                :FB_BA_Label:=( sObjName:='LBL',sDescr:='Blue light intensity');
//     481 BACS sun protection
  LblAgg_BlindAnglePosition                                :FB_BA_Label:=( sObjName:='BAP',sDescr:='Blind angle position');
  LblAgg_ShadingPosition                                   :FB_BA_Label:=( sObjName:='BSP',sDescr:='Shading position');
  LblAgg_MovementCommand                                   :FB_BA_Label:=( sObjName:='BMC',sDescr:='Blind movement command');
//     485 Room automation
  LblAgg_DisplayAndControlUnit                             :FB_BA_Label:=( sObjName:='DCU',sDescr:='Display and control unit');
  LblAgg_PresenceSwitches                                  :FB_BA_Label:=( sObjName:='PDE',sDescr:='Presence switches, detectors, motion detectors');
  LblAgg_RoomAutomationDevice                              :FB_BA_Label:=( sObjName:='RAD',sDescr:='Room automation device');
  LblAgg_RoomControlUnit                                   :FB_BA_Label:=( sObjName:='RCU',sDescr:='Room control unit');
//     Beckhoff ADS communication
  LblAgg_GeneralSettingsCom                                :FB_BA_Label:=( sObjName:='COM',sDescr:='System parameters communication');
  LblAgg_GeneralSettingsComDst                             :FB_BA_Label:=( sObjName:='WEK',sDescr:='Disturbance system parameters communication');
  LblAgg_DataCommunicationExternalControl                  :FB_BA_Label:=( sObjName:='COM',sDescr:='Communication external control');
END_VAR

// ---- Templates/GVLs/Language/English/LblControl_EN.TcGVL
{region '#Template'}
	{attribute 'Version' := '5.1.1.0'}
	{attribute 'Tags' := '"LCID": "1031", "Text": "GVL, AKS, Labels, ObjectName, Description"'}
	{attribute 'Tags' := '"LCID": "1033", "Text": "GVL, DPAD, Labels, ObjectName, Description"'}
	{attribute 'Description' := '"LCID": "1031", "Text": "Anlagenkennzeichnungssystem, Labels controls"'}
	{attribute 'Description' := '"LCID": "1033", "Text": "Data Point Addressing Description, Labels controls"'}
{endregion}
	 
{attribute 'global_init_slot' := '40510'}
VAR_GLOBAL
  LblCtl_OperationMode                                     :FB_BA_Label:=( sObjName:='OPM', sDescr:='Operation mode');
  LblCtl_SummerNightCooling                                :FB_BA_Label:=( sObjName:='SNC', sDescr:='Summer night cooling');
  LblCtl_DifferencePressureMonitoringSupplyAirFan          :FB_BA_Label:=( sObjName:='DPM', sDescr:='Difference pressure monitoring supply air fan');
  LblCtl_DifferencePressureMonitoringExtractAirFan         :FB_BA_Label:=( sObjName:='DPM', sDescr:='Difference pressure monitoring extract air fan');
  LblCtl_TSetpointCalculation                              :FB_BA_Label:=( sObjName:='SPC', sDescr:='Setpoint calculation temperature');
  LblCtl_HSetpointCalculation                              :FB_BA_Label:=( sObjName:='SPC', sDescr:='Setpoint calculation humidity');
  LblCtl_TCascadeSupplyAirControl                          :FB_BA_Label:=( sObjName:='CTL', sDescr:='Cascade control supply air temperature');
  LblCtl_HCascadeSupplyAirControl                          :FB_BA_Label:=( sObjName:='CTL', sDescr:='Cascade control supply air humidity');
  LblCtl_PreHeater                                         :FB_BA_Label:=( sObjName:='PRH', sDescr:='Preheater');
  LblCtl_ReHeater                                          :FB_BA_Label:=( sObjName:='RHE', sDescr:='Reheater');
  LblCtl_EnergyRecovery                                    :FB_BA_Label:=( sObjName:='ERC', sDescr:='Energy recovery');
  LblCtl_SupplyAirTemperatureControl                       :FB_BA_Label:=( sObjName:='CTL', sDescr:='Supply air temperature control');
  LblCtl_SupplyAirDehumidifierControl                      :FB_BA_Label:=( sObjName:='CTL', sDescr:='Supply air dehumidification control');
  LblCtl_SupplyAirHumidifierController                     :FB_BA_Label:=( sObjName:='CTL', sDescr:='Supply air humidity control');
  LblCtl_SupplyAirTemperatureLimitationControl             :FB_BA_Label:=( sObjName:='CTL', sDescr:='Supply air temperature limitation control');
  LblCtl_ReturnWaterControl                                :FB_BA_Label:=( sObjName:='CTL', sDescr:='Return water control');
  LblCtl_HumidityLimitationControl                         :FB_BA_Label:=( sObjName:='CTL', sDescr:='Rel humidity limitation control');
  LblCtl_CalculationPreRinseSetpoint                       :FB_BA_Label:=( sObjName:='SPC', sDescr:='Calculation prerinse setpoint');
  LblCtl_FrostProtectionControl                            :FB_BA_Label:=( sObjName:='FPC', sDescr:='Frost protection control');
  LblCtl_ExhaustAirTemperatureControl                      :FB_BA_Label:=( sObjName:='CTL', sDescr:='Exhaust air temperature control');
  LblCtl_EnergyRecoveryDeicingRamp                         :FB_BA_Label:=( sObjName:='RMP', sDescr:='Energy recovery deicing ramp');
  LblCtl_BACnetDevice                                      :FB_BA_Label:=( sObjName:='DEV', sDescr:='BACnet device');
  LblCtl_PlantControl                                      :FB_BA_Label:=( sObjName:='PCT', sDescr:='Plant control');
  LblCtl_TSequenceControl                                  :FB_BA_Label:=( sObjName:='SEQ', sDescr:='Sequence control temp');
  LblCtl_HSequenceControl                                  :FB_BA_Label:=( sObjName:='SEQ', sDescr:='Sequence control humidity');
  LblCtl_GeneralBeckhoffEventClass                         :FB_BA_Label:=( sObjName:='ECL', sDescr:='Event class');
  LblCtl_GeneralSettings                                   :FB_BA_Label:=( sObjName:='SYP', sDescr:='System parameters');
  LblCtl_GeneralCabinetBasicEquipment                      :FB_BA_Label:=( sObjName:='CBE', sDescr:='Cabinet basic equipment');
  LblCtl_GeneralCabinetAdditionalEquipment                 :FB_BA_Label:=( sObjName:='CAE', sDescr:='Cabinet additional equipment');
  LblCtl_EventIndicationLamp                               :FB_BA_Label:=( sObjName:='CEM', sDescr:='Collective error message lamp');
  LblCtl_AcknowledgeCommand                                :FB_BA_Label:=( sObjName:='ACK', sDescr:='Acknowledge hardware');
  LblCtl_RemoteAcknowledgement                             :FB_BA_Label:=( sObjName:='ACK', sDescr:='Remote acknowledgement fault');
  LblCtl_LocalAcknowledgement                              :FB_BA_Label:=( sObjName:='ACK', sDescr:='Local acknowledgement fault');
  LblCtl_Acknowledge                                       :FB_BA_Label:=( sObjName:='ACK', sDescr:='Acknowledge');
//     
  LblCtl_Fuse                                              :FB_BA_Label:=( sObjName:='FUS', sDescr:='Fuse');
//     Settings
  LblCtl_FrostProtection                                   :FB_BA_Label:=( sObjName:='FRP', sDescr:='Frost protection');
  LblCtl_MinimumOutsideTemperature                         :FB_BA_Label:=( sObjName:='TWT', sDescr:='Minimum outdoor temperature');
  LblCtl_TemperatureWeatherLowLimit                        :FB_BA_Label:=( sObjName:='TWT', sDescr:='Temperature weather low limit');
  LblCtl_TemperatureWeatherDamped                          :FB_BA_Label:=( sObjName:='TWD', sDescr:='Temperature weather damped');
  LblCtl_TemperatureWeatherDampedLowLimit                  :FB_BA_Label:=( sObjName:='TWD', sDescr:='Temperature weather damped low limit');
  LblCtl_PressureControl                                   :FB_BA_Label:=( sObjName:='CTL', sDescr:='Pressure control');
  LblCtl_Converter3Point                                   :FB_BA_Label:=( sObjName:='CNV', sDescr:='3 point converter');
  LblCtl_HeatingCurve                                      :FB_BA_Label:=( sObjName:='HCV', sDescr:='Heating curve');
  LblCtl_SetpointGeneration                                :FB_BA_Label:=( sObjName:='SPG', sDescr:='Setpoint generation');
  LblCtl_RequestHeatState                                  :FB_BA_Label:=( sObjName:='RHS', sDescr:='Request heat state');
  LblCtl_RequestHeatSetpoint                               :FB_BA_Label:=( sObjName:='RHS', sDescr:='Request heat setpoint');
  LblCtl_FlowTempControl                                   :FB_BA_Label:=( sObjName:='CTL', sDescr:='Flow temperature control');
//     
  LblCtl_RoomTemperatureControl                            :FB_BA_Label:=( sObjName:='CTL', sDescr:='Room temperature control');
  LblCtl_FlowTemperatureControl                            :FB_BA_Label:=( sObjName:='CTL', sDescr:='Flow temperature control');
  LblCtl_HeatValve                                         :FB_BA_Label:=( sObjName:='VLV', sDescr:='Heat valve');
  LblCtl_CoolValve                                         :FB_BA_Label:=( sObjName:='VLV', sDescr:='Cool valve');
  LblCtl_HeatingController                                 :FB_BA_Label:=( sObjName:='LPH', sDescr:='Heating controller');
  LblCtl_CoolingController                                 :FB_BA_Label:=( sObjName:='LPC', sDescr:='Cooling controller');
  LblCtl_Light                                             :FB_BA_Label:=( sObjName:='LGT', sDescr:='Light');
  LblCtl_SetpointHeating                                   :FB_BA_Label:=( sObjName:='SPG', sDescr:='Setpoint generation heating');
  LblCtl_SetpointCooling                                   :FB_BA_Label:=( sObjName:='SPG', sDescr:='Setpoint generation cooling');
  LblCtl_Facade                                            :FB_BA_Label:=( sObjName:='FIE', sDescr:='Facade data');
  LblCtl_BuildingAlarms                                    :FB_BA_Label:=( sObjName:='FIE', sDescr:='Building alarms');
  LblCtl_BuildingEnergyLevel                               :FB_BA_Label:=( sObjName:='FIE', sDescr:='Building energylevel');
  LblCtl_BuildingMode                                      :FB_BA_Label:=( sObjName:='FIE', sDescr:='Building operationmode');
  LblCtl_BuildingSpRmT                                     :FB_BA_Label:=( sObjName:='FIE', sDescr:='Building roomtemperature setpoints');
  LblCtl_BuildingSunprotection                             :FB_BA_Label:=( sObjName:='FIE', sDescr:='Building sunprotection');
  LblCtl_TemperatureFrost                                  :FB_BA_Label:=( sObjName:='TFR', sDescr:='Temperature frost');
  LblCtl_MixedAirStartUpRamp                               :FB_BA_Label:=( sObjName:='RMP', sDescr:='Ramp plant start');
  LblCtl_Cooler                                            :FB_BA_Label:=( sObjName:='COL', sDescr:='Cooler');
  LblCtl_EvtCategoryLifeSafty                              :FB_BA_Label:=( sObjName:='EDL', sDescr:='Danger to life');
  LblCtl_EvtCategorySaftyMessage                           :FB_BA_Label:=( sObjName:='ESM', sDescr:='Safety message');
  LblCtl_EvtCategoryAlarmMessage                           :FB_BA_Label:=( sObjName:='EAM', sDescr:='Alarm message');
  LblCtl_EvtCategoryFaultMessage                           :FB_BA_Label:=( sObjName:='EFM', sDescr:='Fault message');
  LblCtl_EvtCategoryMaintenanceMessage                     :FB_BA_Label:=( sObjName:='EMM', sDescr:='Maintenance message');
  LblCtl_EvtCategorySystem                                 :FB_BA_Label:=( sObjName:='ESY', sDescr:='System message');
  LblCtl_EvtCategoryManualOperation                        :FB_BA_Label:=( sObjName:='EMO', sDescr:='Manual operation');
  LblCtl_EvtCategoryOther                                  :FB_BA_Label:=( sObjName:='EOM', sDescr:='Other message');
  LblCtl_TrendLogging                                      :FB_BA_Label:=( sObjName:='TRL', sDescr:='');
  LblCtl_WeatherParameters                                 :FB_BA_Label:=( sObjName:='WTP', sDescr:='Weather parameters');
  LblCtl_SetpointFrostProtection                           :FB_BA_Label:=( sObjName:='SP_', sDescr:='Setpoint frost protection');
  LblCtl_SetpointWeatherIcing                              :FB_BA_Label:=( sObjName:='SP_', sDescr:='Setpoint icing');
  LblCtl_SetpointMinimumOutsideTemperature                 :FB_BA_Label:=( sObjName:='SPI', sDescr:='Setpoint minimum outside temperature');
  LblCtl_MeanDamped                                        :FB_BA_Label:=( sObjName:='MWD', sDescr:='Mean value weather temperature damped');
  LblCtl_OperationalMessageTemperatureWeatherLowLimit      :FB_BA_Label:=( sObjName:='OM_', sDescr:='Operational message temperature weather low limit');
  LblCtl_OperationalMessageTemperatureWeatherDampedLowLimit:FB_BA_Label:=( sObjName:='OM_', sDescr:='Operational message temperature weather damped low limit');
  LblCtl_PlantStartup                                      :FB_BA_Label:=( sObjName:='PST', sDescr:='Plant startup');
  LblCtl_TimeDelayDampersClose                             :FB_BA_Label:=( sObjName:='TD_', sDescr:='Time delay dampers close, fans run down');
  LblCtl_TimeDelaySupplyAirFanOn                           :FB_BA_Label:=( sObjName:='TD_', sDescr:='Time delay supply air fan on');
  LblCtl_TimeDelayExtractAirFanOn                          :FB_BA_Label:=( sObjName:='TD_', sDescr:='Time delay extract air fan on');
  LblCtl_TimeDelayTemperatureSequenceControlOn             :FB_BA_Label:=( sObjName:='TD_', sDescr:='Time delay temperature sequence control on');
  LblCtl_TimeDelayTemperatureSequenceControlOff            :FB_BA_Label:=( sObjName:='TD_', sDescr:='Time delay temperature sequence control off');
  LblCtl_TimeDelayHumiditySequenceControlOn                :FB_BA_Label:=( sObjName:='TD_', sDescr:='Time delay humidity sequence control on');
  LblCtl_TimeDelayEnableMonitoringLimitValues              :FB_BA_Label:=( sObjName:='TD_', sDescr:='Time delay enable monitoring limit values');
  LblCtl_StagesOfThePlantStartup                           :FB_BA_Label:=( sObjName:='STA', sDescr:='Stages of the plant startup');
//     Beckhoff cabinet basic equipment
  LblCtl_SwitchingCommandCollectiveFaultSignalLamp         :FB_BA_Label:=( sObjName:='SC_', sDescr:='Collective fault signal lamp switching command');
  LblCtl_SwitchingCommandHardwareAcknowledgement           :FB_BA_Label:=( sObjName:='SC_', sDescr:='Hardware acknowledgement switching command');
  LblCtl_ButtonRemoteAcknowledgement                       :FB_BA_Label:=( sObjName:='BUT', sDescr:='Input remote acknowledgement');
  LblCtl_ButtonLocalAcknowledgement                        :FB_BA_Label:=( sObjName:='BUT', sDescr:='Button acknowledgement');
//     Beckhoff heating circuit
  LblCtl_HeatingLimit                                      :FB_BA_Label:=( sObjName:='HLM', sDescr:='Heating limit ');
  LblCtl_PresentOperationMode                              :FB_BA_Label:=( sObjName:='POM', sDescr:='Present operation mode');
  LblCtl_OperationModeSelection                            :FB_BA_Label:=( sObjName:='OMS', sDescr:='Operation mode selection');
//     Beckhoff summer night cooling
  LblCtl_HysteresisRoomTemperature                         :FB_BA_Label:=( sObjName:='HYS', sDescr:='Hysteresis room temperature');
  LblCtl_OutsideTemperatureLowLimit                        :FB_BA_Label:=( sObjName:='MIN', sDescr:='Minimum outside temperature');
  LblCtl_OffValueDifferenceOutsideInsightTemperature       :FB_BA_Label:=( sObjName:='MIN', sDescr:='Off value difference between ouside and insight temperature');
  LblCtl_OnValueDifferenceOutsideInsightTemperature        :FB_BA_Label:=( sObjName:='MAX', sDescr:='On value difference between ouside and insight temperature');
//     Beckhoff damper
  LblCtl_DriveTimeOpen                                     :FB_BA_Label:=( sObjName:='DTO', sDescr:='Drive time open');
  LblCtl_DriveTimeClose                                    :FB_BA_Label:=( sObjName:='DTC', sDescr:='Drive time close');
  LblCtl_DisturbanceFeedbackOpen                           :FB_BA_Label:=( sObjName:='DSO', sDescr:='Disturbance feedback open');
  LblCtl_DisturbanceFeedbackClose                          :FB_BA_Label:=( sObjName:='DSC', sDescr:='Disturbance feedback close');
//     
  LblCtl_TimeDelay                                         :FB_BA_Label:=( sObjName:='TD_', sDescr:='Time delay ');
  LblCtl_TimeDelayFeedback                                 :FB_BA_Label:=( sObjName:='TDF', sDescr:='Time delay feedback');
  LblCtl_TimeDelayInterruptionFeedback                     :FB_BA_Label:=( sObjName:='TDI', sDescr:='Time delay interruption');
//     Beckhoff prerinse
  LblCtl_PreRinseDuration                                  :FB_BA_Label:=( sObjName:='PRD', sDescr:='Prerinse duration');
  LblCtl_DisturbancePreRinse                               :FB_BA_Label:=( sObjName:='DST', sDescr:='Disturbance prerinse');
  LblCtl_SetpointMinimalReturnWaterTemperature             :FB_BA_Label:=( sObjName:='SP_', sDescr:='Setpoint minimal return water temperature');
//     Beckhoff ramp 
  LblCtl_RampTimeUp                                        :FB_BA_Label:=( sObjName:='RTU', sDescr:='Ramp time up');
  LblCtl_RampTimeDown                                      :FB_BA_Label:=( sObjName:='RTD', sDescr:='Ramp time down');
  LblCtl_CommandOpen                                       :FB_BA_Label:=( sObjName:='SC_', sDescr:='Switch command open');
  LblCtl_CommandClose                                      :FB_BA_Label:=( sObjName:='SC_', sDescr:='Switch command close');
  LblCtl_CalculatedValue                                   :FB_BA_Label:=( sObjName:='CAV', sDescr:='Calculated value');
  LblCtl_Value                                             :FB_BA_Label:=( sObjName:='VAL', sDescr:='Value');
//     Beckhoff event class
  LblCtl_EvtClass                                          :FB_BA_Label:=( sObjName:='NC_', sDescr:='Notification class');
  LblCtl_FlowSwitch                                        :FB_BA_Label:=( sObjName:='OM_', sDescr:='Operating message flow monitor');
  LblCtl_SmokeAlarm                                        :FB_BA_Label:=( sObjName:='DST', sDescr:='Disturbance smoke alarm');
  LblCtl_SystemFailure                                     :FB_BA_Label:=( sObjName:='DST', sDescr:='Disturbance system failure');
  LblCtl_Contamination                                     :FB_BA_Label:=( sObjName:='DST', sDescr:='Disturbance contamination');
  LblCtl_SwitchingCommandSmokeDetector                     :FB_BA_Label:=( sObjName:='SC_', sDescr:='Switching command acknowledge');
  LblCtl_ButtonReset                                       :FB_BA_Label:=( sObjName:='BUT', sDescr:='Button acknowledge');
  LblCtl_OffsetNightSetpoint                               :FB_BA_Label:=( sObjName:='ONS', sDescr:='Offset night setback');
//     
  LblCtl_SetpointRelHumidityHumidification                 :FB_BA_Label:=( sObjName:='SP_', sDescr:='Setpoint relative humidity humidification');
  LblCtl_SetpointRelHumidityDehumidification               :FB_BA_Label:=( sObjName:='SP_', sDescr:='Setpoint relative humidity dehumidification');
  LblCtl_SetpointAbsHumidityHumidification                 :FB_BA_Label:=( sObjName:='SPC', sDescr:='Setpoint absolute humidity humidification');
  LblCtl_SetpointAbsHumidityDehumidification               :FB_BA_Label:=( sObjName:='SPC', sDescr:='Setpoint absolute humidity dehumidification');
  LblCtl_SetpointRelHumidity                               :FB_BA_Label:=( sObjName:='SP_', sDescr:='Setpoint relative humidity');
  LblCtl_SetpointAbsHumidity                               :FB_BA_Label:=( sObjName:='SP_', sDescr:='Setpoint absolute humidity');
  LblCtl_OperationalMessageDehumidification                :FB_BA_Label:=( sObjName:='OM_', sDescr:='Operational message dehumidification');
//     
  LblCtl_SetpointSunblindPosition                          :FB_BA_Label:=( sObjName:='SP_', sDescr:='Setpoint blind position');
  LblCtl_SetpointSunblindAngle                             :FB_BA_Label:=( sObjName:='SP_', sDescr:='Setpoint blind angle');
  LblCtl_CommandSunblindStart                              :FB_BA_Label:=( sObjName:='SC_', sDescr:='Command sunblind start');
  LblCtl_ButtonSunblind                                    :FB_BA_Label:=( sObjName:='BUT', sDescr:='Sun blind button');
  LblCtl_FeedbackSunblindPosition                          :FB_BA_Label:=( sObjName:='FDB', sDescr:='Feedback blind position');
  LblCtl_FeedbackSunblindAngle                             :FB_BA_Label:=( sObjName:='FDB', sDescr:='Feedback blind angle');
  LblCtl_FeedbackSunblindPrio                              :FB_BA_Label:=( sObjName:='FDB', sDescr:='Feedback telegram-priority');
//     
  LblCtl_TimeDelayStormOn                                  :FB_BA_Label:=( sObjName:='TON', sDescr:='Storm-detection time delay on');
  LblCtl_TimeDelayStormOff                                 :FB_BA_Label:=( sObjName:='TOF', sDescr:='Storm-detection time delay off');
  LblCtl_MaintenanceEnable                                 :FB_BA_Label:=( sObjName:='EN_', sDescr:='Maintenence positioning enable');
  LblCtl_MaintenancePosition                               :FB_BA_Label:=( sObjName:='SP_', sDescr:='Setpoint maintenance position');
  LblCtl_MaintenanceAngle                                  :FB_BA_Label:=( sObjName:='SP_', sDescr:='Setpoint maintenance angle');
  LblCtl_FacadeThermoAutomaticEnable                       :FB_BA_Label:=( sObjName:='EN_', sDescr:='Facade-thermoautomatic enable');
  LblCtl_FacadeThermoAutomaticCoolingPosition              :FB_BA_Label:=( sObjName:='SP_', sDescr:='Facade-thermoautomatic cooling-position');
  LblCtl_FacadeThermoAutomaticCoolingAngle                 :FB_BA_Label:=( sObjName:='SP_', sDescr:='Facade-thermoautomatic cooling-angle');
  LblCtl_FacadeTwilightAutomaticEnable                     :FB_BA_Label:=( sObjName:='EN_', sDescr:='Facade-twilightautomatic enable');
  LblCtl_SunProtectionValueOn                              :FB_BA_Label:=( sObjName:='SP_', sDescr:='Sun-protection brightness on');
  LblCtl_SunProtectionValueOn0deg                          :FB_BA_Label:=( sObjName:='SP_', sDescr:='Sun-protection brightness on at elevation 0 deg');
  LblCtl_SunProtectionValueOn15deg                         :FB_BA_Label:=( sObjName:='SP_', sDescr:='Sun-protection brightness on at elevation 15 deg');
  LblCtl_SunProtectionValueOn30deg                         :FB_BA_Label:=( sObjName:='SP_', sDescr:='Sun-protection brightness on at elevation 30 deg');
  LblCtl_SunProtectionValueOn45deg                         :FB_BA_Label:=( sObjName:='SP_', sDescr:='Sun-protection brightness on at elevation 45 deg');
  LblCtl_SunProtectionValueOn60deg                         :FB_BA_Label:=( sObjName:='SP_', sDescr:='Sun-protection brightness on at elevation 60 deg');
  LblCtl_SunProtectionValueOn75deg                         :FB_BA_Label:=( sObjName:='SP_', sDescr:='Sun-protection brightness on at elevation 75 deg');
  LblCtl_SunProtectionValueOn90deg                         :FB_BA_Label:=( sObjName:='SP_', sDescr:='Sun-protection brightness on at elevation 90 deg');
  LblCtl_SunProtectionValueOff                             :FB_BA_Label:=( sObjName:='SP_', sDescr:='Sun-protection brightness off');
  LblCtl_SunProtectionValueOff0deg                         :FB_BA_Label:=( sObjName:='SP_', sDescr:='Sun-protection brightness off at elevation 0 deg');
  LblCtl_SunProtectionValueOff15deg                        :FB_BA_Label:=( sObjName:='SP_', sDescr:='Sun-protection brightness off at elevation 15 deg');
  LblCtl_SunProtectionValueOff30deg                        :FB_BA_Label:=( sObjName:='SP_', sDescr:='Sun-protection brightness off at elevation 30 deg');
  LblCtl_SunProtectionValueOff45deg                        :FB_BA_Label:=( sObjName:='SP_', sDescr:='Sun-protection brightness off at elevation 45 deg');
  LblCtl_SunProtectionValueOff60deg                        :FB_BA_Label:=( sObjName:='SP_', sDescr:='Sun-protection brightness off at elevation 60 deg');
  LblCtl_SunProtectionValueOff75deg                        :FB_BA_Label:=( sObjName:='SP_', sDescr:='Sun-protection brightness off at elevation 75 deg');
  LblCtl_SunProtectionValueOff90deg                        :FB_BA_Label:=( sObjName:='SP_', sDescr:='Sun-protection brightness off at elevation 90 deg');
  LblCtl_TimeDelaySunProtectionOn                          :FB_BA_Label:=( sObjName:='TON', sDescr:='Sun-protection brightness on');
  LblCtl_TimeDelaySunProtectionOff                         :FB_BA_Label:=( sObjName:='TOF', sDescr:='Sun-protection brightness off');
  LblCtl_FacadeParkingEnable                               :FB_BA_Label:=( sObjName:='EN_', sDescr:='Facade-parking enable');
  LblCtl_FacadeParkingPosition                             :FB_BA_Label:=( sObjName:='SP_', sDescr:='Facade-parking position');
  LblCtl_FacadeParkingAngle                                :FB_BA_Label:=( sObjName:='SP_', sDescr:='Facade-parking angle');
  LblCtl_WindProtectionState                               :FB_BA_Label:=( sObjName:='STA', sDescr:='State wind-protection');
  LblCtl_SunProtectionState                                :FB_BA_Label:=( sObjName:='STA', sDescr:='State sun-protection');
  LblCtl_WindProtection                                    :FB_BA_Label:=( sObjName:='WPR', sDescr:='Windprotection');
  LblCtl_Maintenance                                       :FB_BA_Label:=( sObjName:='MTC', sDescr:='Maintenance');
  LblCtl_ThermoAutomatic                                   :FB_BA_Label:=( sObjName:='THA', sDescr:='Thermoautomatic');
  LblCtl_TwilightAutomatic                                 :FB_BA_Label:=( sObjName:='TWA', sDescr:='Twilightautomatic');
  LblCtl_Parking                                           :FB_BA_Label:=( sObjName:='PAK', sDescr:='Parking');
  LblCtl_SunProtection                                     :FB_BA_Label:=( sObjName:='SUN', sDescr:='Sunprotection');
  LblCtl_FacadeInformation                                 :FB_BA_Label:=( sObjName:='FIN', sDescr:='Facade-information');
  LblCtl_PrioResultingTelegram                             :FB_BA_Label:=( sObjName:='PFT', sDescr:='Priority actual facade-telegram');
  LblCtl_SunProtectionValueOnCalc                          :FB_BA_Label:=( sObjName:='SPC', sDescr:='Calculated brightness-limit sunprotection on');
  LblCtl_SunProtectionValueOffCalc                         :FB_BA_Label:=( sObjName:='SPC', sDescr:='Calculated brightness-limit sunprotection off');
  LblCtl_SunblindZoneControl                               :FB_BA_Label:=( sObjName:='SZC', sDescr:='SunBlind zone-control');
  LblCtl_SunblindActuator                                  :FB_BA_Label:=( sObjName:='SBA', sDescr:='Sunblind-actuator');
//     
  LblCtl_LowWaterMonitor                                   :FB_BA_Label:=( sObjName:='DST', sDescr:='Low water monitor');
  LblCtl_FireAlert                                         :FB_BA_Label:=( sObjName:='DST', sDescr:='Fire alert');
  LblCtl_Burglary                                          :FB_BA_Label:=( sObjName:='DST', sDescr:='Burglary alert');
  LblCtl_CentralSwitchOff                                  :FB_BA_Label:=( sObjName:='PLS', sDescr:='Central switch-off');
  LblCtl_ForcedVentilation                                 :FB_BA_Label:=( sObjName:='PLS', sDescr:='Forced ventilation ');
  LblCtl_SmokeExtraction                                   :FB_BA_Label:=( sObjName:='PLS', sDescr:='Smoke extraction');
  LblCtl_SetpointIce                                       :FB_BA_Label:=( sObjName:='SP_', sDescr:='Setpoint ice');
  LblCtl_SunProtectionInterval                             :FB_BA_Label:=( sObjName:='SPI', sDescr:='Sun-protection positioning interval');
  LblCtl_DeiceTime                                         :FB_BA_Label:=( sObjName:='SP_', sDescr:='Frost-protection deice-time');
  LblCtl_GlobalThermoAutomaticValueOn                      :FB_BA_Label:=( sObjName:='SP_', sDescr:='Thermo-automatic radiation-value on');
  LblCtl_GlobalThermoAutomaticValueOff                     :FB_BA_Label:=( sObjName:='SP_', sDescr:='Thermo-automatic radiation-value off');
  LblCtl_GlobalTwilightAutomaticValueOn                    :FB_BA_Label:=( sObjName:='SP_', sDescr:='Twilight-automatic brightness-value on');
  LblCtl_GlobalTwilightAutomaticValueOff                   :FB_BA_Label:=( sObjName:='SP_', sDescr:='Twilight-automatic brightness-value on');
  LblCtl_IceAlert                                          :FB_BA_Label:=( sObjName:='DST', sDescr:='Ice alert');
  LblCtl_MagneticSwitch                                    :FB_BA_Label:=( sObjName:='MGS', sDescr:='Magnetic switch');
  LblCtl_FireDetector                                      :FB_BA_Label:=( sObjName:='FDT', sDescr:='Fire-detector');
  LblCtl_IceProtection                                     :FB_BA_Label:=( sObjName:='IPR', sDescr:='Ice-protection');
  LblCtl_GlobalThermoAutomaticRelease                      :FB_BA_Label:=( sObjName:='EN_', sDescr:='Thermoautomatic release');
  LblCtl_RadiationOn                                       :FB_BA_Label:=( sObjName:='SP_', sDescr:='Radiation value on');
  LblCtl_RadiationOff                                      :FB_BA_Label:=( sObjName:='SP_', sDescr:='Radiation value off');
  LblCtl_RadiationDlyOn                                    :FB_BA_Label:=( sObjName:='TON', sDescr:='Radiation delay on');
  LblCtl_RadiationDlyOff                                   :FB_BA_Label:=( sObjName:='TOF', sDescr:='Radiation delay off');
  LblCtl_GlobalTwilightAutomaticRelease                    :FB_BA_Label:=( sObjName:='EN_', sDescr:='Twilightautomatic release');
  LblCtl_BrightnessOn                                      :FB_BA_Label:=( sObjName:='SP_', sDescr:='Brightness value on');
  LblCtl_BrightnessOff                                     :FB_BA_Label:=( sObjName:='SP_', sDescr:='Brightness value off');
  LblCtl_BrightnessDlyOn                                   :FB_BA_Label:=( sObjName:='TON', sDescr:='Brightness delay on');
  LblCtl_BrightnessDlyOff                                  :FB_BA_Label:=( sObjName:='TOF', sDescr:='Brightness delay off');
  LblCtl_GlobalResetManMode                                :FB_BA_Label:=( sObjName:='PLS', sDescr:='Global reset manual mode');
  LblCtl_GlobalResetLighting                               :FB_BA_Label:=( sObjName:='PLS', sDescr:='Global reset lighting');
  LblCtl_MaintenanceLighting                               :FB_BA_Label:=( sObjName:='PLS', sDescr:='Maintenance switch lighting');
//     
  LblCtl_BuildingEnergyLevelManual                         :FB_BA_Label:=( sObjName:='OPS', sDescr:='Building-energy-level manual selection');
  LblCtl_BuildingEnergyLevelActual                         :FB_BA_Label:=( sObjName:='POM', sDescr:='Building-energy-level actual selection');
  LblCtl_RoomAutomTimeSchedules                            :FB_BA_Label:=( sObjName:='RAT', sDescr:='Room-automation time-schedules');
  LblCtl_BuildingEnergyLevelSched                          :FB_BA_Label:=( sObjName:='SCH', sDescr:='Building-energy-level scheduler');
  LblCtl_BuildingModeManual                                :FB_BA_Label:=( sObjName:='OPS', sDescr:='Building-mode manual selection');
  LblCtl_BuildingModeActual                                :FB_BA_Label:=( sObjName:='POM', sDescr:='Building-mode actual selection');
  LblCtl_BuildingModeSched                                 :FB_BA_Label:=( sObjName:='SCH', sDescr:='Building-mode scheduler');
//     
  LblCtl_SummerCompensationX1                              :FB_BA_Label:=( sObjName:='IPX', sDescr:='Summercompensation X1');
  LblCtl_SummerCompensationX2                              :FB_BA_Label:=( sObjName:='IPX', sDescr:='Summercompensation X2');
  LblCtl_SummerCompensationY1                              :FB_BA_Label:=( sObjName:='IPY', sDescr:='Summercompensation Y1');
  LblCtl_SummerCompensationY2                              :FB_BA_Label:=( sObjName:='IPY', sDescr:='Summercompensation Y2');
  LblCtl_WinterCompensationX1                              :FB_BA_Label:=( sObjName:='IPX', sDescr:='Wintercompensation X1');
  LblCtl_WinterCompensationX2                              :FB_BA_Label:=( sObjName:='IPX', sDescr:='Wintercompensation X2');
  LblCtl_WinterCompensationY1                              :FB_BA_Label:=( sObjName:='IPY', sDescr:='Wintercompensation Y1');
  LblCtl_WinterCompensationY2                              :FB_BA_Label:=( sObjName:='IPY', sDescr:='Wintercompensation Y2');
  LblCtl_SummerCompensation                                :FB_BA_Label:=( sObjName:='SCP', sDescr:='Summercompensation');
  LblCtl_WinterCompensation                                :FB_BA_Label:=( sObjName:='WCP', sDescr:='Wintercompensation');
  LblCtl_SummerCompensationYmin                            :FB_BA_Label:=( sObjName:='SPI', sDescr:='Summer compensation Ymin');
  LblCtl_SummerCompensationYmax                            :FB_BA_Label:=( sObjName:='SPX', sDescr:='Summer compensation Ymax');
  LblCtl_WinterCompensationYmin                            :FB_BA_Label:=( sObjName:='SPI', sDescr:='Winter compensation Ymin');
  LblCtl_WinterCompensationYmax                            :FB_BA_Label:=( sObjName:='SPX', sDescr:='Winter compensation Ymax');
  LblCtl_SummerCompensationSp                              :FB_BA_Label:=( sObjName:='SPC', sDescr:='Summer compensation setpoint');
  LblCtl_WinterCompensationSp                              :FB_BA_Label:=( sObjName:='SPC', sDescr:='Winter compensation setpoint');
  LblCtl_SetpointShiftHeating                              :FB_BA_Label:=( sObjName:='SP_', sDescr:='Setpoint shift heating');
  LblCtl_SetpointShiftCooling                              :FB_BA_Label:=( sObjName:='SP_', sDescr:='Setpoint shift cooling');
  LblCtl_DampConstant                                      :FB_BA_Label:=( sObjName:='SP_', sDescr:='Damp constant');
//     
  LblCtl_DelayOn                                           :FB_BA_Label:=( sObjName:='TON', sDescr:='Switch-on delay');
  LblCtl_DelayOff                                          :FB_BA_Label:=( sObjName:='TOF', sDescr:='Switch-off delay');
  LblCtl_AntiBlocking                                      :FB_BA_Label:=( sObjName:='ABK', sDescr:='Anti blocking');
  LblCtl_IdlePeriod                                        :FB_BA_Label:=( sObjName:='ITV', sDescr:='Idle period');
  LblCtl_ImpulsLength                                      :FB_BA_Label:=( sObjName:='IPL', sDescr:='Impulse length');
  LblCtl_SuppyAirTempSetpointCalc                          :FB_BA_Label:=( sObjName:='SPC', sDescr:='Suppy air setpoint calc');
  LblCtl_SuppyAirTempSetpointHeaterCalc                    :FB_BA_Label:=( sObjName:='SPC', sDescr:='Suppy air setpoint heater calc');
  LblCtl_SuppyAirTempSetpointCoolerCalc                    :FB_BA_Label:=( sObjName:='SPC', sDescr:='Suppy air setpoint cooler calc');
  LblCtl_SuppyAirTempSetpointERCCalc                       :FB_BA_Label:=( sObjName:='SPC', sDescr:='Suppy air setpoint erc calc');
  LblCtl_X01                                               :FB_BA_Label:=( sObjName:='SPX', sDescr:='Value base [X1]');
  LblCtl_X02                                               :FB_BA_Label:=( sObjName:='SPX', sDescr:='Value base [X2]');
  LblCtl_X03                                               :FB_BA_Label:=( sObjName:='SPX', sDescr:='Value base [X3]');
  LblCtl_X04                                               :FB_BA_Label:=( sObjName:='SPX', sDescr:='Value base [X4]');
  LblCtl_X05                                               :FB_BA_Label:=( sObjName:='SPX', sDescr:='Value base [X5]');
  LblCtl_X06                                               :FB_BA_Label:=( sObjName:='SPX', sDescr:='Value base [X6]');
  LblCtl_X07                                               :FB_BA_Label:=( sObjName:='SPX', sDescr:='Value base [X7]');
  LblCtl_Y01                                               :FB_BA_Label:=( sObjName:='SPY', sDescr:='Value base [Y1]');
  LblCtl_Y02                                               :FB_BA_Label:=( sObjName:='SPY', sDescr:='Value base [Y2]');
  LblCtl_Y02_03                                            :FB_BA_Label:=( sObjName:='SPY', sDescr:='Value base [Y2Y3]');
  LblCtl_Y03                                               :FB_BA_Label:=( sObjName:='SPY', sDescr:='Value base [Y3]');
  LblCtl_Y04                                               :FB_BA_Label:=( sObjName:='SPY', sDescr:='Value base [Y4]');
  LblCtl_Y05                                               :FB_BA_Label:=( sObjName:='SPY', sDescr:='Value base [Y5]');
  LblCtl_Y06                                               :FB_BA_Label:=( sObjName:='SPY', sDescr:='Value base [Y6]');
  LblCtl_Y07                                               :FB_BA_Label:=( sObjName:='SPY', sDescr:='Value base [Y7]');
  LblCtl_FeedbackMonitoring                                :FB_BA_Label:=( sObjName:='FDM', sDescr:='Feedback monitoring');
  LblCtl_PreAlarmLimitMAX                                  :FB_BA_Label:=( sObjName:='LMX', sDescr:='Pre alarm limit max');
  LblCtl_PreAlarmLimitMIN                                  :FB_BA_Label:=( sObjName:='LMI', sDescr:='Pre alarm limit min');
  LblCtl_PreAlarmFault                                     :FB_BA_Label:=( sObjName:='DST', sDescr:='Pre alarm fault');
  LblCtl_MainAlarmLimitMAX                                 :FB_BA_Label:=( sObjName:='LMX', sDescr:='Main alarm limit max');
  LblCtl_MainAlarmLimitMIN                                 :FB_BA_Label:=( sObjName:='LMI', sDescr:='Main alarm limit min');
  LblCtl_MainAlarmFault                                    :FB_BA_Label:=( sObjName:='DST', sDescr:='Main alarm fault');
  LblCtl_ProcPreRinse                                      :FB_BA_LabelProcess:=( sProcessName:='Process prerinse');
  LblCtl_ProjectInfo                                       :FB_BA_Label:=( sObjName:='PI_', sDescr:='Project info');
//     
  LblCtl_BrightnessPresenceSensor                          :FB_BA_Label:=( sObjName:='BPS', sDescr:='Brightness-and presence-sensor');
  LblCtl_BuildingLighting                                  :FB_BA_Label:=( sObjName:='FIE', sDescr:='Building light control');
  LblCtl_SetpointLightValue                                :FB_BA_Label:=( sObjName:='SP_', sDescr:='Setpoint light-value');
  LblCtl_SetpointLightTemperature                          :FB_BA_Label:=( sObjName:='SP_', sDescr:='Setpoint light-temperature');
  LblCtl_SetpointBrightness                                :FB_BA_Label:=( sObjName:='SP_', sDescr:='Setpoint brightness');
  LblCtl_FeedbackLightValue                                :FB_BA_Label:=( sObjName:='FDB', sDescr:='Feedback light-value');
  LblCtl_FeedbackLightTemperature                          :FB_BA_Label:=( sObjName:='FDB', sDescr:='Feedback light-temperature');
  LblCtl_FeedbackLightPrio                                 :FB_BA_Label:=( sObjName:='FDB', sDescr:='Feedback priority of light-telegram');
  LblCtl_ButtonLight                                       :FB_BA_Label:=( sObjName:='BUT', sDescr:='Light-switch');
  LblCtl_LightBuilding                                     :FB_BA_Label:=( sObjName:='LBD', sDescr:='Light-control building');
  LblCtl_LightFloor                                        :FB_BA_Label:=( sObjName:='LFL', sDescr:='Light-control floor');
  LblCtl_LightArea                                         :FB_BA_Label:=( sObjName:='LAR', sDescr:='Light-control area');
  LblCtl_LightZoneControl                                  :FB_BA_Label:=( sObjName:='LZC', sDescr:='Light zone-control');
  LblCtl_LightActuator                                     :FB_BA_Label:=( sObjName:='LAC', sDescr:='Light-actuator');
  LblCtl_SetpointLightValueCleaning                        :FB_BA_Label:=( sObjName:='SP_', sDescr:='Setpoint light-value cleaning');
  LblCtl_SetpointLightTemperatureCleaning                  :FB_BA_Label:=( sObjName:='SP_', sDescr:='Setpoint light-temperature cleaning');
  LblCtl_SetpointLightValueNightwatch                      :FB_BA_Label:=( sObjName:='SP_', sDescr:='Setpoint light-value nightwatch');
  LblCtl_SetpointLightTemperatureNightwatch                :FB_BA_Label:=( sObjName:='SP_', sDescr:='Setpoint light-temperature nightwatch');
  LblCtl_SetpointLightValueMaintenance                     :FB_BA_Label:=( sObjName:='SP_', sDescr:='Setpoint light-value maintenance');
  LblCtl_SetpointLightTemperatureMaintenance               :FB_BA_Label:=( sObjName:='SP_', sDescr:='Setpoint light-temperature maintenance');
  LblCtl_SetpointLightValueUserDefined1                    :FB_BA_Label:=( sObjName:='SP_', sDescr:='Setpoint light-value user-defined 1');
  LblCtl_SetpointLightTemperatureUserDefined1              :FB_BA_Label:=( sObjName:='SP_', sDescr:='Setpoint light-temperature user-defined 1');
  LblCtl_SetpointLightValueUserDefined2                    :FB_BA_Label:=( sObjName:='SP_', sDescr:='Setpoint light-value user-defined 2');
  LblCtl_SetpointLightTemperatureUserDefined2              :FB_BA_Label:=( sObjName:='SP_', sDescr:='Setpoint light-temperature user-defined 2');
//     
  LblCtl_LimitValueWeatherTemperatureSummer                :FB_BA_Label:=( sObjName:='LM_', sDescr:='Limit value weather temperature summer');
  LblCtl_LimitValueWeatherTemperatureWinter                :FB_BA_Label:=( sObjName:='LM_', sDescr:='Limit value weather temperature winter');
  LblCtl_CurrentSequenceTemperature                        :FB_BA_Label:=( sObjName:='STA', sDescr:='Current sequence temperature');
  LblCtl_CurrentSequenceHumidity                           :FB_BA_Label:=( sObjName:='STA', sDescr:='Current sequence humidity');
  LblCtl_DeviceWeatherStationDataDisturbed                 :FB_BA_Label:=( sObjName:='DST', sDescr:='Device weatherstation-data disturbed');
  LblCtl_DeviceGeneralDataDisturbed                        :FB_BA_Label:=( sObjName:='DST', sDescr:='Device general data disturbed');
  LblCtl_DeviceBuildingEnergyLevelDisturbed                :FB_BA_Label:=( sObjName:='DST', sDescr:='Device building-energy-level-disturbed');
  LblCtl_DeviceBuildingModeDisturbed                       :FB_BA_Label:=( sObjName:='DST', sDescr:='Device building-mode-data disturbed');
  LblCtl_DeviceBuildingSunBlindDataDisturbed               :FB_BA_Label:=( sObjName:='DST', sDescr:='Device building-sunblind-data disturbed');
  LblCtl_DeviceBuildingAlarmsDisturbed                     :FB_BA_Label:=( sObjName:='DST', sDescr:='Device building-alarms disturbed');
  LblCtl_DeviceBuildingSpRmTDisturbed                      :FB_BA_Label:=( sObjName:='DST', sDescr:='Device buildingwide roomtemperature-setpoints disturbed');
  LblCtl_DeviceBuildingLightingDataDisturbed               :FB_BA_Label:=( sObjName:='DST', sDescr:='Device building-lighting-data disturbed');
  LblCtl_Facade1CommunicationDisturbance                   :FB_BA_Label:=( sObjName:='DST', sDescr:='Facade 1 communication disturbed');
  LblCtl_Facade2CommunicationDisturbance                   :FB_BA_Label:=( sObjName:='DST', sDescr:='Facade 2 communication disturbed');
  LblCtl_Facade3CommunicationDisturbance                   :FB_BA_Label:=( sObjName:='DST', sDescr:='Facade 3 communication disturbed');
  LblCtl_Facade4CommunicationDisturbance                   :FB_BA_Label:=( sObjName:='DST', sDescr:='Facade 4 communication disturbed');
END_VAR

// ---- Templates/GVLs/Language/English/LblFunctions_EN.TcGVL
{region '#Template'}
	{attribute 'Version' := '5.0.0.0'}
	{attribute 'Tags' := '"LCID": "1031", "Text": "GVL, AKS, Labels, ObjectName, Description"'}
	{attribute 'Tags' := '"LCID": "1033", "Text": "GVL, DPAD, Labels, ObjectName, Description"'}
	{attribute 'Description' := '"LCID": "1031", "Text": "Anlagenkennzeichnungssystem, Labels functions"'}
	{attribute 'Description' := '"LCID": "1033", "Text": "Data Point Addressing Description, Labels functions"'}
{endregion}

